KUKA KRL program: MyProgram_237().src

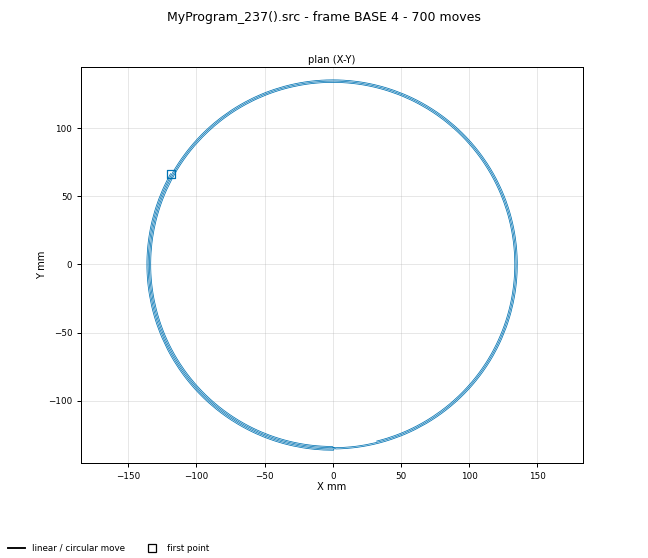
[picture p0: tool path of MyProgram_237().src in frame BASE 4, 700 of 700 moves have a stored position in this frame; points joined in program order, loops and branches not executed]
&ACCESS RVP
&REL 1
&PARAM TEMPLATE = C:\KRC\Roboter\Template\vorgabe
&PARAM EDITMASK = *
DEF MyProgram_237()
; ---- Setting reference (Base) ----
$BASE = BASE_DATA[4]

; --------------------------
; ---- Setting tool (TCP) ----
$TOOL = TOOL_DATA[3]
; --------------------------

$VEL.CP = VEL_APROX_PRINT
Startdeposition()
$VEL.CP = VEL_PRINT
LIN {X -118.9926,Y 66.6239,Z 160,A 148.5784,B 23.5572,C -1.283,E1 23.449,E2 298.3688} C_DIS
LIN {X -121.2876,Y 62.3465,Z 160,A 150.2313,B 23.5584,C -1.2585,E1 23.447,E2 296.7681} C_DIS
LIN {X -123.5569,Y 57.7188,Z 160,A 152.2779,B 23.5591,C -1.2464,E1 23.4445,E2 294.7403} C_DIS
LIN {X -125.0146,Y 54.4885,Z 160,A 153.7,B 23.5594,C -1.2386,E1 23.4429,E2 293.3293} C_DIS
LIN {X -126.4544,Y 51.0566,Z 160,A 155.2792,B 23.5596,C -1.2346,E1 23.4412,E2 291.751} C_DIS
LIN {X -127.5918,Y 48.145,Z 160,A 156.5985,B 23.5598,C -1.2307,E1 23.4399,E2 290.4334} C_DIS
LIN {X -128.7443,Y 44.9722,Z 160,A 158.0153,B 23.5601,C -1.2262,E1 23.4386,E2 289.0194} C_DIS
LIN {X -129.5584,Y 42.5724,Z 160,A 159.5184,B 23.5592,C -1.2435,E1 23.4373,E2 287.4635} C_DIS
LIN {X -130.7224,Y 38.8522,Z 160,A 160.8124,B 23.5603,C -1.2221,E1 23.4362,E2 286.2155} C_DIS
LIN {X -131.707,Y 35.3675,Z 160,A 162.2633,B 23.5607,C -1.2139,E1 23.4352,E2 284.7762} C_DIS
LIN {X -132.5011,Y 32.2662,Z 160,A 163.6223,B 23.5608,C -1.2102,E1 23.4342,E2 283.4179} C_DIS
LIN {X -133.2335,Y 29.0944,Z 160,A 165.0699,B 23.5608,C -1.2096,E1 23.4334,E2 281.9629} C_DIS
LIN {X -134.0169,Y 25.2423,Z 160,A 166.7918,B 23.561,C -1.2075,E1 23.4324,E2 280.2352} C_DIS
LIN {X -134.7535,Y 20.9542,Z 160,A 168.5433,B 23.5614,C -1.198,E1 23.4317,E2 278.4967} C_DIS
LIN {X -135.3189,Y 16.9412,Z 160,A 170.3698,B 23.5614,C -1.1982,E1 23.431,E2 276.658} C_DIS
LIN {X -135.712,Y 13.4163,Z 160,A 171.719,B 23.562,C -1.1867,E1 23.4306,E2 275.329} C_DIS
LIN {X -136.0044,Y 10.0208,Z 160,A 173.2395,B 23.562,C -1.1862,E1 23.4303,E2 273.8} C_DIS
LIN {X -136.2543,Y 5.7048,Z 160,A 175.0307,B 23.5623,C -1.1791,E1 23.43,E2 272.0153} C_DIS
LIN {X -136.3568,Y 2.1131,Z 160,A 176.588,B 23.5624,C -1.1764,E1 23.43,E2 270.4546} C_DIS
LIN {X -136.3514,Y -2.4394,Z 160,A 178.4811,B 23.5628,C -1.1693,E1 23.43,E2 268.5674} C_DIS
LIN {X -136.2184,Y -6.5022,Z 160,A -179.7767,B 23.563,C -1.1653,E1 23.4302,E2 266.8239} C_DIS
LIN {X -135.9819,Y -10.3286,Z 160,A -178.1684,B 23.5632,C -1.16,E1 23.4305,E2 265.2187} C_DIS
LIN {X -135.6069,Y -14.4357,Z 160,A -176.4169,B 23.5634,C -1.1553,E1 23.4309,E2 263.4679} C_DIS
LIN {X -135.1517,Y -18.2164,Z 160,A -174.7244,B 23.5634,C -1.1545,E1 23.4315,E2 261.7665} C_DIS
LIN {X -134.5594,Y -22.1676,Z 160,A -173.1183,B 23.5639,C -1.1457,E1 23.4322,E2 260.1723} C_DIS
LIN {X -132.9907,Y -30.1838,Z 160,A -169.6362,B 23.5643,C -1.1372,E1 23.4342,E2 256.6896} C_DIS
LIN {X -132.0789,Y -33.9538,Z 160,A -167.9215,B 23.5643,C -1.1361,E1 23.4354,E2 254.9669} C_DIS
LIN {X -130.964,Y -38.0269,Z 160,A -166.3432,B 23.565,C -1.1214,E1 23.4365,E2 253.4161} C_DIS
LIN {X -130.0625,Y -41.0063,Z 160,A -164.8722,B 23.5648,C -1.1251,E1 23.4378,E2 251.9266} C_DIS
LIN {X -128.9154,Y -44.4789,Z 160,A -163.3824,B 23.5651,C -1.1182,E1 23.4391,E2 250.445} C_DIS
LIN {X -127.7244,Y -47.7909,Z 160,A -161.9393,B 23.5654,C -1.1121,E1 23.4405,E2 249.0086} C_DIS
LIN {X -126.5403,Y -50.8435,Z 160,A -160.482,B 23.5654,C -1.1119,E1 23.442,E2 247.5431} C_DIS
LIN {X -125.2476,Y -53.9495,Z 160,A -159.1344,B 23.5657,C -1.1047,E1 23.4434,E2 246.2057} C_DIS
LIN {X -121.1191,Y -62.6761,Z 160,A -155.0024,B 23.5661,C -1.0965,E1 23.4485,E2 242.0702} C_DIS
LIN {X -118.6948,Y -67.1543,Z 160,A -152.7589,B 23.5661,C -1.0956,E1 23.4515,E2 239.8165} C_DIS
LIN {X -116.5618,Y -70.7914,Z 160,A -151.0585,B 23.5665,C -1.0874,E1 23.4539,E2 238.1273} C_DIS
LIN {X -112.5394,Y -77.0255,Z 160,A -147.8415,B 23.5666,C -1.084,E1 23.4588,E2 234.9016} C_DIS
LIN {X -109.8378,Y -80.8311,Z 160,A -145.9935,B 23.5671,C -1.0736,E1 23.4618,E2 233.0701} C_DIS
LIN {X -107.641,Y -83.7346,Z 160,A -144.404,B 23.5671,C -1.0728,E1 23.4645,E2 231.4747} C_DIS
LIN {X -104.9293,Y -87.1084,Z 160,A -142.6985,B 23.5675,C -1.0629,E1 23.4675,E2 229.7855} C_DIS
LIN {X -101.6155,Y -90.9522,Z 160,A -140.3512,B 23.5673,C -1.0684,E1 23.4719,E2 227.4131} C_DIS
LIN {X -98.4957,Y -94.3219,Z 160,A -138.5662,B 23.5678,C -1.0571,E1 23.4753,E2 225.6482} C_DIS
LIN {X -94.701,Y -98.1314,Z 160,A -136.1362,B 23.5676,C -1.0605,E1 23.4801,E2 223.1987} C_DIS
LIN {X -91.0992,Y -101.4838,Z 160,A -133.1464,B 23.5658,C -1.1018,E1 23.4866,E2 220.0923} C_DIS
LIN {X -85.5869,Y -106.1739,Z 160,A -131.0457,B 23.5681,C -1.0495,E1 23.4908,E2 218.1147} C_DIS
LIN {X -81.7858,Y -109.1296,Z 160,A -129.0308,B 23.5683,C -1.0454,E1 23.4953,E2 216.1021} C_DIS
LIN {X -78.2738,Y -111.6754,Z 160,A -127.1485,B 23.5683,C -1.0452,E1 23.4996,E2 214.2134} C_DIS
LIN {X -74.6255,Y -114.1456,Z 160,A -125.3166,B 23.5684,C -1.0412,E1 23.5038,E2 212.385} C_DIS
LIN {X -69.3964,Y -117.398,Z 160,A -122.6893,B 23.5685,C -1.0393,E1 23.5101,E2 209.7539} C_DIS
LIN {X -66.0931,Y -119.2884,Z 160,A -121.1313,B 23.5687,C -1.035,E1 23.5139,E2 208.2019} C_DIS
LIN {X -62.2401,Y -121.3417,Z 160,A -119.3539,B 23.5689,C -1.0298,E1 23.5183,E2 206.4324} C_DIS
LIN {X -59.0874,Y -122.9075,Z 160,A -117.8743,B 23.5689,C -1.028,E1 23.522,E2 204.9531} C_DIS
LIN {X -55.9819,Y -124.3528,Z 160,A -116.6382,B 23.5695,C -1.0162,E1 23.5251,E2 203.7433} C_DIS
LIN {X -50.5222,Y -126.6698,Z 160,A -113.9638,B 23.5692,C -1.0226,E1 23.532,E2 201.0463} C_DIS
LIN {X -46.435,Y -128.2237,Z 160,A -112.0439,B 23.5692,C -1.025,E1 23.5371,E2 199.1161} C_DIS
LIN {X -42.7262,Y -129.5072,Z 160,A -110.3745,B 23.5692,C -1.0247,E1 23.5415,E2 197.4442} C_DIS
LIN {X -38.5738,Y -130.8039,Z 160,A -108.6083,B 23.5693,C -1.0202,E1 23.5462,E2 195.686} C_DIS
LIN {X -35.2796,Y -131.7304,Z 160,A -107.2059,B 23.5694,C -1.0175,E1 23.5499,E2 194.2881} C_DIS
LIN {X -31.7741,Y -132.6197,Z 160,A -105.6159,B 23.5694,C -1.0202,E1 23.5543,E2 192.689} C_DIS
LIN {X -28.5037,Y -133.361,Z 160,A -103.3189,B 23.5674,C -1.0649,E1 23.5609,E2 190.277} C_DIS
LIN {X -21.8819,Y -134.6071,Z 160,A -101.3405,B 23.5693,C -1.0202,E1 23.566,E2 188.4086} C_DIS
LIN {X -17.9115,Y -135.1917,Z 160,A -99.972,B 23.57,C -1.0037,E1 23.5697,E2 187.0802} C_DIS
LIN {X -12.7092,Y -135.7799,Z 160,A -96.6912,B 23.5677,C -1.0589,E1 23.5792,E2 183.6593} C_DIS
LIN {X -6.5196,Y -136.2175,Z 160,A -94.9524,B 23.5696,C -1.0141,E1 23.5837,E2 182.0318} C_DIS
LIN {X 0.6255,Y -136.3718,Z 160,A -92.0832,B 23.5698,C -1.0077,E1 23.5917,E2 179.1785} C_DIS
LIN {X 0.6255,Y -136.3718,Z 160,A -92.0832,B 23.5698,C -1.0077,E1 23.5917,E2 179.1785} C_DIS
Enddeposition()
LIN {X 0.9621,Y -135.4362,Z 160,A -91.6873,B 21.9641,C -0.7399,E1 21.9772,E2 179.2938} C_DIS
Startdeposition()
$VEL.CP = VEL_PRINT
LIN {X -3.6024,Y -135.3994,Z 160,A -93.5739,B 21.9641,C -0.7415,E1 21.9719,E2 181.1761} C_DIS
LIN {X -6.6447,Y -135.2842,Z 160,A -95.1252,B 21.9644,C -0.7291,E1 21.9675,E2 182.761} C_DIS
LIN {X -10.3175,Y -135.0544,Z 160,A -96.9624,B 21.9649,C -0.7161,E1 21.9623,E2 184.6339} C_DIS
LIN {X -13.5627,Y -134.7677,Z 160,A -98.238,B 21.9647,C -0.721,E1 21.9587,E2 185.8972} C_DIS
LIN {X -17.8068,Y -134.2716,Z 160,A -99.829,B 21.9644,C -0.7314,E1 21.9544,E2 187.4617} C_DIS
LIN {X -21.1498,Y -133.7863,Z 160,A -101.2751,B 21.9644,C -0.731,E1 21.9504,E2 188.9102} C_DIS
LIN {X -24.2668,Y -133.256,Z 160,A -102.9482,B 21.9649,C -0.716,E1 21.9457,E2 190.6255} C_DIS
LIN {X -27.6501,Y -132.5963,Z 160,A -104.0571,B 21.9643,C -0.7327,E1 21.9428,E2 191.6912} C_DIS
LIN {X -30.692,Y -131.9248,Z 160,A -105.4462,B 21.9644,C -0.7301,E1 21.939,E2 193.0893} C_DIS
LIN {X -34.7695,Y -130.9082,Z 160,A -107.2187,B 21.9644,C -0.7314,E1 21.9342,E2 194.8612} C_DIS
LIN {X -38.1022,Y -129.9772,Z 160,A -108.6616,B 21.9644,C -0.7333,E1 21.9303,E2 196.3015} C_DIS
LIN {X -41.3625,Y -128.9767,Z 160,A -110.1289,B 21.9644,C -0.7333,E1 21.9264,E2 197.7719} C_DIS
LIN {X -45.0409,Y -127.7405,Z 160,A -112.0238,B 21.9646,C -0.7232,E1 21.9213,E2 199.6982} C_DIS
LIN {X -49.2765,Y -126.1653,Z 160,A -113.6914,B 21.9642,C -0.7361,E1 21.917,E2 201.3352} C_DIS
LIN {X -55.4887,Y -123.5591,Z 160,A -116.5223,B 21.9641,C -0.74,E1 21.9098,E2 204.1632} C_DIS
LIN {X -58.5818,Y -122.1229,Z 160,A -117.9831,B 21.9641,C -0.7409,E1 21.9061,E2 205.626} C_DIS
LIN {X -61.723,Y -120.566,Z 160,A -119.474,B 21.9641,C -0.7424,E1 21.9024,E2 207.1174} C_DIS
LIN {X -65.1604,Y -118.7458,Z 160,A -121.2225,B 21.9641,C -0.7399,E1 21.898,E2 208.8782} C_DIS
LIN {X -69.084,Y -116.506,Z 160,A -123.512,B 21.9645,C -0.7258,E1 21.8924,E2 211.2135} C_DIS
LIN {X -72.7665,Y -114.243,Z 160,A -124.6697,B 21.9635,C -0.7585,E1 21.8899,E2 212.2876} C_DIS
LIN {X -75.1993,Y -112.6561,Z 160,A -126.1897,B 21.9639,C -0.7475,E1 21.8862,E2 213.8431} C_DIS
LIN {X -78.8618,Y -110.1234,Z 160,A -128.0645,B 21.9637,C -0.751,E1 21.882,E2 215.7158} C_DIS
LIN {X -82.5025,Y -107.4231,Z 160,A -130.0066,B 21.9637,C -0.7533,E1 21.8776,E2 217.6598} C_DIS
LIN {X -85.9062,Y -104.7211,Z 160,A -131.8112,B 21.9635,C -0.7582,E1 21.8737,E2 219.459} C_DIS
LIN {X -90.4175,Y -100.8514,Z 160,A -134.3556,B 21.9634,C -0.7618,E1 21.8684,E2 222.0053} C_DIS
LIN {X -93.6344,Y -97.8719,Z 160,A -136.2177,B 21.9633,C -0.7653,E1 21.8646,E2 223.8669} C_DIS
LIN {X -97.1401,Y -94.3938,Z 160,A -138.3591,B 21.9633,C -0.7675,E1 21.8603,E2 226.0129} C_DIS
LIN {X -100.2567,Y -91.0765,Z 160,A -140.2831,B 21.9631,C -0.7718,E1 21.8567,E2 227.9351} C_DIS
LIN {X -103.4388,Y -87.4464,Z 160,A -142.1169,B 21.9626,C -0.7856,E1 21.8534,E2 229.7413} C_DIS
LIN {X -105.4457,Y -85.0148,Z 160,A -143.6687,B 21.9628,C -0.7792,E1 21.8506,E2 231.3186} C_DIS
LIN {X -108.2907,Y -81.3606,Z 160,A -145.6019,B 21.9626,C -0.7851,E1 21.8473,E2 233.2467} C_DIS
LIN {X -110.878,Y -77.7979,Z 160,A -147.5162,B 21.9626,C -0.7875,E1 21.8442,E2 235.1653} C_DIS
LIN {X -113.242,Y -74.3143,Z 160,A -149.4657,B 21.9626,C -0.7848,E1 21.8412,E2 237.1335} C_DIS
LIN {X -115.5765,Y -70.6289,Z 160,A -151.1544,B 21.9622,C -0.7964,E1 21.8387,E2 238.8009} C_DIS
LIN {X -117.8279,Y -66.806,Z 160,A -153.1467,B 21.9622,C -0.7964,E1 21.8359,E2 240.8051} C_DIS
LIN {X -120.0606,Y -62.7002,Z 160,A -154.9729,B 21.9618,C -0.8084,E1 21.8336,E2 242.6103} C_DIS
LIN {X -121.9143,Y -59.0186,Z 160,A -157.2735,B 21.9625,C -0.7893,E1 21.8307,E2 244.9767} C_DIS
LIN {X -123.878,Y -54.7756,Z 160,A -158.6627,B 21.9614,C -0.8202,E1 21.8292,E2 246.2915} C_DIS
LIN {X -125.0588,Y -52.0206,Z 160,A -159.9812,B 21.9614,C -0.8217,E1 21.8277,E2 247.6144} C_DIS
LIN {X -126.3506,Y -48.7999,Z 160,A -161.4648,B 21.9612,C -0.8253,E1 21.8262,E2 249.098} C_DIS
LIN {X -127.5141,Y -45.6733,Z 160,A -162.8651,B 21.961,C -0.8299,E1 21.8249,E2 250.4949} C_DIS
LIN {X -128.731,Y -42.1266,Z 160,A -164.5953,B 21.961,C -0.8284,E1 21.8233,E2 252.2406} C_DIS
LIN {X -129.9198,Y -38.2981,Z 160,A -166.2639,B 21.9609,C -0.8347,E1 21.822,E2 253.9034} C_DIS
LIN {X -130.9593,Y -34.5776,Z 160,A -167.8267,B 21.9606,C -0.8428,E1 21.8208,E2 255.455} C_DIS
LIN {X -132.0465,Y -30.1591,Z 160,A -170.7115,B 21.9618,C -0.808,E1 21.819,E2 258.4531} C_DIS
LIN {X -133.3797,Y -23.5757,Z 160,A -172.5089,B 21.9599,C -0.8611,E1 21.8181,E2 260.1197} C_DIS
LIN {X -133.8391,Y -20.8086,Z 160,A -173.8181,B 21.9599,C -0.8596,E1 21.8175,E2 261.442} C_DIS
LIN {X -134.3147,Y -17.4777,Z 160,A -175.2975,B 21.9599,C -0.8617,E1 21.8169,E2 262.9261} C_DIS
LIN {X -134.8037,Y -13.1884,Z 160,A -177.1458,B 21.9597,C -0.8665,E1 21.8164,E2 264.7741} C_DIS
LIN {X -135.1311,Y -9.2669,Z 160,A -178.8967,B 21.9597,C -0.8681,E1 21.816,E2 266.5329} C_DIS
LIN {X -135.3485,Y -5.1699,Z 160,A 179.4466,B 21.9593,C -0.8771,E1 21.8158,E2 268.1771} C_DIS
LIN {X -135.4457,Y -0.789,Z 160,A 177.6628,B 21.959,C -0.886,E1 21.8158,E2 269.9493} C_DIS
LIN {X -135.4241,Y 2.5173,Z 160,A 176.1951,B 21.959,C -0.8875,E1 21.8158,E2 271.4231} C_DIS
LIN {X -135.2841,Y 6.6458,Z 160,A 174.4162,B 21.9587,C -0.8918,E1 21.816,E2 273.2028} C_DIS
LIN {X -135.06,Y 10.2409,Z 160,A 172.8421,B 21.9587,C -0.8945,E1 21.8163,E2 274.7805} C_DIS
LIN {X -134.6705,Y 14.4832,Z 160,A 171.1093,B 21.9583,C -0.9033,E1 21.8168,E2 276.5017} C_DIS
LIN {X -134.2709,Y 17.8124,Z 160,A 169.6786,B 21.9581,C -0.9073,E1 21.8173,E2 277.9315} C_DIS
LIN {X -133.724,Y 21.5484,Z 160,A 167.9141,B 21.9582,C -0.9053,E1 21.818,E2 279.7136} C_DIS
LIN {X -133.0318,Y 25.4642,Z 160,A 166.3272,B 21.9578,C -0.9147,E1 21.8188,E2 281.286} C_DIS
LIN {X -132.1863,Y 29.5473,Z 160,A 164.4073,B 21.9578,C -0.9137,E1 21.8199,E2 283.2218} C_DIS
LIN {X -131.2621,Y 33.4084,Z 160,A 162.8919,B 21.9574,C -0.926,E1 21.8209,E2 284.7143} C_DIS
LIN {X -130.1663,Y 37.4562,Z 160,A 160.6198,B 21.958,C -0.9104,E1 21.8227,E2 287.0436} C_DIS
LIN {X -128.9607,Y 41.4127,Z 160,A 159.3216,B 21.957,C -0.935,E1 21.8238,E2 288.2841} C_DIS
LIN {X -127.974,Y 44.3677,Z 160,A 158.0167,B 21.9568,C -0.9396,E1 21.8249,E2 289.5853} C_DIS
LIN {X -126.7763,Y 47.6825,Z 160,A 156.5194,B 21.9567,C -0.9439,E1 21.8264,E2 291.0807} C_DIS
LIN {X -125.5135,Y 50.9143,Z 160,A 155.041,B 21.9565,C -0.9479,E1 21.8279,E2 292.5579} C_DIS
LIN {X -124.2359,Y 53.9564,Z 160,A 153.597,B 21.9565,C -0.9501,E1 21.8295,E2 294.0053} C_DIS
LIN {X -122.6045,Y 57.5724,Z 160,A 151.6607,B 21.9567,C -0.9441,E1 21.8318,E2 295.9701} C_DIS
LIN {X -120.4337,Y 61.9828,Z 160,A 149.8245,B 21.956,C -0.9606,E1 21.834,E2 297.7732} C_DIS
LIN {X -117.8067,Y 66.8432,Z 160,A 147.3938,B 21.9559,C -0.9633,E1 21.8373,E2 300.2113} C_DIS
LIN {X -115.6401,Y 70.5253,Z 160,A 145.5271,B 21.9558,C -0.9659,E1 21.84,E2 302.0822} C_DIS
LIN {X -113.1582,Y 74.4416,Z 160,A 143.2602,B 21.9561,C -0.9584,E1 21.8435,E2 304.3827} C_DIS
LIN {X -110.9089,Y 77.754,Z 160,A 142.1606,B 21.9548,C -0.9884,E1 21.8452,E2 305.4077} C_DIS
LIN {X -107.9092,Y 81.8661,Z 160,A 139.6213,B 21.9553,C -0.9776,E1 21.8494,E2 307.9903} C_DIS
LIN {X -105.2413,Y 85.2682,Z 160,A 137.3826,B 21.9558,C -0.9648,E1 21.8534,E2 310.2753} C_DIS
LIN {X -102.1389,Y 88.9605,Z 160,A 135.9969,B 21.9544,C -0.9981,E1 21.8558,E2 311.5789} C_DIS
LIN {X -99.6611,Y 91.7278,Z 160,A 134.2543,B 21.9545,C -0.9946,E1 21.8591,E2 313.3398} C_DIS
LIN {X -96.5021,Y 95.0461,Z 160,A 132.3015,B 21.9544,C -0.9987,E1 21.8629,E2 315.2915} C_DIS
LIN {X -93.3021,Y 98.1896,Z 160,A 130.3884,B 21.9542,C -1.0025,E1 21.8667,E2 317.2035} C_DIS
LIN {X -90.0635,Y 101.1684,Z 160,A 128.5201,B 21.954,C -1.0064,E1 21.8706,E2 319.0699} C_DIS
LIN {X -86.7543,Y 104.0201,Z 160,A 125.8575,B 21.9554,C -0.9753,E1 21.8765,E2 321.8278} C_DIS
LIN {X -81.7211,Y 108.0185,Z 160,A 124.1711,B 21.9532,C -1.0257,E1 21.88,E2 323.386} C_DIS
LIN {X -74.5587,Y 113.0811,Z 160,A 120.1563,B 21.9534,C -1.0196,E1 21.8892,E2 327.4329} C_DIS
LIN {X -71.1893,Y 115.2326,Z 160,A 118.4924,B 21.9533,C -1.0239,E1 21.8931,E2 329.0914} C_DIS
LIN {X -67.4456,Y 117.463,Z 160,A 116.6616,B 21.9531,C -1.0277,E1 21.8975,E2 330.9183} C_DIS
LIN {X -63.8987,Y 119.4292,Z 160,A 114.9581,B 21.9529,C -1.0311,E1 21.9017,E2 332.6183} C_DIS
LIN {X -59.1266,Y 121.8627,Z 160,A 112.7618,B 21.9526,C -1.0378,E1 21.9072,E2 334.8034} C_DIS
LIN {X -56.6,Y 123.0541,Z 160,A 111.5172,B 21.9526,C -1.0368,E1 21.9103,E2 336.0541} C_DIS
LIN {X -52.5123,Y 124.8534,Z 160,A 109.4998,B 21.9528,C -1.0339,E1 21.9155,E2 338.085} C_DIS
LIN {X -49.0701,Y 126.2456,Z 160,A 108.0641,B 21.9525,C -1.0419,E1 21.9192,E2 339.5027} C_DIS
LIN {X -45.7417,Y 127.4895,Z 160,A 106.6127,B 21.9523,C -1.0461,E1 21.923,E2 340.9462} C_DIS
LIN {X -42.5303,Y 128.5966,Z 160,A 105.1147,B 21.9523,C -1.0451,E1 21.927,E2 342.4502} C_DIS
LIN {X -35.6562,Y 130.6717,Z 160,A 102.1237,B 21.9521,C -1.0504,E1 21.935,E2 345.4328} C_DIS
LIN {X -31.5859,Y 131.7126,Z 160,A 100.2958,B 21.9521,C -1.0498,E1 21.9399,E2 347.2652} C_DIS
LIN {X -27.3973,Y 132.6477,Z 160,A 98.4634,B 21.9521,C -1.0506,E1 21.9449,E2 349.0983} C_DIS
LIN {X -23.7948,Y 133.3405,Z 160,A 96.9896,B 21.9518,C -1.0552,E1 21.949,E2 350.5612} C_DIS
LIN {X -20.6085,Y 133.8701,Z 160,A 95.5687,B 21.9519,C -1.0537,E1 21.9529,E2 351.9878} C_DIS
LIN {X -17.0008,Y 134.3772,Z 160,A 93.9024,B 21.9521,C -1.0489,E1 21.9575,E2 353.6683} C_DIS
LIN {X -12.6352,Y 134.8568,Z 160,A 92.1536,B 21.9519,C -1.0548,E1 21.9624,E2 355.4026} C_DIS
LIN {X -8.3244,Y 135.1911,Z 160,A 90.3503,B 21.9518,C -1.0567,E1 21.9674,E2 357.2016} C_DIS
LIN {X -4.4468,Y 135.3759,Z 160,A 88.5636,B 21.9521,C -1.0506,E1 21.9724,E2 359.0051} C_DIS
LIN {X 0.0544,Y 135.449,Z 160,A 86.661,B 21.9521,C -1.051,E1 21.9777,E2 360.9065} C_DIS
LIN {X 3.8844,Y 135.3915,Z 160,A 85.1395,B 21.9518,C -1.0557,E1 21.9819,E2 362.4151} C_DIS
LIN {X 8.0031,Y 135.2109,Z 160,A 83.2602,B 21.9521,C -1.0495,E1 21.9872,E2 364.3103} C_DIS
LIN {X 13.1417,Y 134.8082,Z 160,A 81.2144,B 21.9518,C -1.0554,E1 21.9929,E2 366.3389} C_DIS
LIN {X 17.6346,Y 134.2942,Z 160,A 79.2629,B 21.9519,C -1.0532,E1 21.9983,E2 368.2945} C_DIS
LIN {X 21.6033,Y 133.7149,Z 160,A 77.4061,B 21.9523,C -1.0453,E1 22.0035,E2 370.1705} C_DIS
LIN {X 26.0559,Y 132.9187,Z 160,A 75.5996,B 21.9521,C -1.0494,E1 22.0084,E2 371.9637} C_DIS
LIN {X 30.0594,Y 132.0693,Z 160,A 73.9772,B 21.9519,C -1.0535,E1 22.0128,E2 373.5724} C_DIS
LIN {X 33.4396,Y 131.2542,Z 160,A 72.5493,B 21.9519,C -1.0546,E1 22.0166,E2 374.995} C_DIS
LIN {X 36.6391,Y 130.3973,Z 160,A 71.1278,B 21.9519,C -1.0527,E1 22.0204,E2 376.4189} C_DIS
LIN {X 40.1258,Y 129.3678,Z 160,A 69.5912,B 21.952,C -1.0516,E1 22.0246,E2 377.9553} C_DIS
LIN {X 45.1696,Y 127.6957,Z 160,A 67.366,B 21.952,C -1.0507,E1 22.0304,E2 380.178} C_DIS
LIN {X 52.3518,Y 124.9205,Z 160,A 64.1027,B 21.9522,C -1.0471,E1 22.0389,E2 383.4425} C_DIS
LIN {X 55.4472,Y 123.5776,Z 160,A 62.6685,B 21.9523,C -1.0451,E1 22.0426,E2 384.8779} C_DIS
LIN {X 58.6262,Y 122.1017,Z 160,A 61.1812,B 21.9523,C -1.0431,E1 22.0463,E2 386.3661} C_DIS
LIN {X 61.8215,Y 120.5158,Z 160,A 59.6981,B 21.9524,C -1.0424,E1 22.05,E2 387.8466} C_DIS
LIN {X 65.2203,Y 118.7131,Z 160,A 57.957,B 21.9528,C -1.0347,E1 22.0544,E2 389.6023} C_DIS
LIN {X 69.1222,Y 116.484,Z 160,A 56.0779,B 21.9528,C -1.0329,E1 22.0589,E2 391.4794} C_DIS
LIN {X 72.8604,Y 114.1829,Z 160,A 54.2455,B 21.9529,C -1.0312,E1 22.0632,E2 393.3098} C_DIS
LIN {X 76.4861,Y 111.7866,Z 160,A 52.3879,B 21.9531,C -1.0273,E1 22.0675,E2 395.1706} C_DIS
LIN {X 80.3614,Y 109.034,Z 160,A 50.5718,B 21.9528,C -1.0331,E1 22.0716,E2 396.9639} C_DIS
LIN {X 83.2733,Y 106.8271,Z 160,A 48.0827,B 21.9549,C -0.9853,E1 22.0773,E2 399.5697} C_DIS
LIN {X 88.1924,Y 102.8032,Z 160,A 46.3323,B 21.9532,C -1.0248,E1 22.0808,E2 401.2069} C_DIS
LIN {X 90.926,Y 100.3933,Z 160,A 44.6612,B 21.9536,C -1.0155,E1 22.0843,E2 402.8953} C_DIS
LIN {X 94.8811,Y 96.6639,Z 160,A 42.7284,B 21.9531,C -1.0284,E1 22.0882,E2 404.7845} C_DIS
LIN {X 97.6299,Y 93.8877,Z 160,A 40.6857,B 21.9541,C -1.0059,E1 22.0923,E2 406.877} C_DIS
LIN {X 101.7299,Y 89.4287,Z 160,A 38.2535,B 21.9541,C -1.0064,E1 22.0968,E2 409.2954} C_DIS
LIN {X 104.372,Y 86.3297,Z 160,A 36.4603,B 21.9544,C -0.9989,E1 22.1,E2 411.099} C_DIS
LIN {X 107.206,Y 82.7844,Z 160,A 34.5509,B 21.9545,C -0.9948,E1 22.1033,E2 413.009} C_DIS
LIN {X 109.9242,Y 79.1402,Z 160,A 31.9269,B 21.9562,C -0.956,E1 22.1078,E2 415.7214} C_DIS
LIN {X 113.3162,Y 74.2015,Z 160,A 30.1356,B 21.9549,C -0.9855,E1 22.1104,E2 417.424} C_DIS
LIN {X 115.6843,Y 70.4532,Z 160,A 28.2272,B 21.9552,C -0.979,E1 22.1132,E2 419.3386} C_DIS
LIN {X 117.9534,Y 66.5838,Z 160,A 26.3474,B 21.9554,C -0.9747,E1 22.1158,E2 421.2186} C_DIS
LIN {X 120.0672,Y 62.6878,Z 160,A 24.593,B 21.9554,C -0.9755,E1 22.1181,E2 422.9602} C_DIS
LIN {X 121.5296,Y 59.8027,Z 160,A 23.2355,B 21.9554,C -0.9722,E1 22.1198,E2 424.3181} C_DIS
LIN {X 123.0606,Y 56.5858,Z 160,A 21.7446,B 21.9556,C -0.9687,E1 22.1216,E2 425.8089} C_DIS
LIN {X 124.3792,Y 53.625,Z 160,A 20.3817,B 21.9558,C -0.9652,E1 22.1231,E2 427.1726} C_DIS
LIN {X 125.7532,Y 50.3195,Z 160,A 18.7788,B 21.9562,C -0.9564,E1 22.1248,E2 428.7887} C_DIS
LIN {X 127.1636,Y 46.6454,Z 160,A 17.1142,B 21.9564,C -0.9515,E1 22.1265,E2 430.4557} C_DIS
LIN {X 128.9475,Y 41.4541,Z 160,A 14.5207,B 21.9572,C -0.9312,E1 22.1288,E2 433.0862} C_DIS
LIN {X 130.073,Y 37.7751,Z 160,A 13.3187,B 21.9565,C -0.9472,E1 22.1297,E2 434.2376} C_DIS
LIN {X 130.975,Y 34.5191,Z 160,A 11.7596,B 21.957,C -0.9364,E1 22.1308,E2 435.8151} C_DIS
LIN {X 132.0121,Y 30.3097,Z 160,A 10.0128,B 21.957,C -0.9351,E1 22.1319,E2 437.5537} C_DIS
LIN {X 132.7768,Y 26.763,Z 160,A 8.5324,B 21.9571,C -0.933,E1 22.1328,E2 439.0297} C_DIS
LIN {X 133.5293,Y 22.7156,Z 160,A 6.7512,B 21.9574,C -0.9256,E1 22.1337,E2 440.8186} C_DIS
LIN {X 134.0985,Y 19.0657,Z 160,A 5.2345,B 21.9575,C -0.9229,E1 22.1343,E2 442.3321} C_DIS
LIN {X 134.6344,Y 14.8184,Z 160,A 3.4079,B 21.9578,C -0.9164,E1 22.1349,E2 444.1636} C_DIS
LIN {X 134.9855,Y 11.1757,Z 160,A 1.9516,B 21.9578,C -0.916,E1 22.1353,E2 445.6108} C_DIS
LIN {X 135.3137,Y 6.0543,Z 160,A -0.1724,B 21.958,C -0.9114,E1 22.1356,E2 447.7326} C_DIS
LIN {X 135.438,Y 1.6818,Z 160,A -2.0292,B 21.9582,C -0.9051,E1 22.1357,E2 449.5932} C_DIS
LIN {X 135.4206,Y -2.7263,Z 160,A -3.9036,B 21.9585,C -0.8986,E1 22.1357,E2 451.4721} C_DIS
LIN {X 135.3312,Y -5.6134,Z 160,A -5.2414,B 21.9588,C -0.8889,E1 22.1355,E2 452.8264} C_DIS
LIN {X 135.0829,Y -9.9261,Z 160,A -6.9508,B 21.9588,C -0.8889,E1 22.1352,E2 454.5241} C_DIS
LIN {X 134.7869,Y -13.3631,Z 160,A -8.3674,B 21.9589,C -0.8863,E1 22.1349,E2 455.9379} C_DIS
LIN {X 134.3342,Y -17.3291,Z 160,A -10.1624,B 21.9594,C -0.8756,E1 22.1343,E2 457.7492} C_DIS
LIN {X 133.8352,Y -20.8335,Z 160,A -11.5719,B 21.9594,C -0.8752,E1 22.1337,E2 459.1502} C_DIS
LIN {X 133.2551,Y -24.2722,Z 160,A -13.1368,B 21.9597,C -0.866,E1 22.1329,E2 460.729} C_DIS
LIN {X 132.4172,Y -28.488,Z 160,A -14.8303,B 21.9597,C -0.8664,E1 22.132,E2 462.41} C_DIS
LIN {X 131.6464,Y -31.8606,Z 160,A -16.2421,B 21.9597,C -0.8643,E1 22.1311,E2 463.8178} C_DIS
LIN {X 130.8612,Y -34.9456,Z 160,A -17.6089,B 21.96,C -0.859,E1 22.1301,E2 465.1896} C_DIS
LIN {X 129.8924,Y -38.3919,Z 160,A -19.1189,B 21.9601,C -0.8545,E1 22.1289,E2 466.7017} C_DIS
LIN {X 128.3314,Y -43.3267,Z 160,A -21.2591,B 21.9603,C -0.8501,E1 22.1271,E2 468.8395} C_DIS
LIN {X 127.2422,Y -46.4275,Z 160,A -23.545,B 21.962,C -0.8015,E1 22.1248,E2 471.2397} C_DIS
LIN {X 124.9157,Y -52.3633,Z 160,A -24.9813,B 21.9601,C -0.8557,E1 22.1235,E2 472.5229} C_DIS
LIN {X 123.9701,Y -54.5686,Z 160,A -26.3438,B 21.9609,C -0.8352,E1 22.1219,E2 473.9312} C_DIS
LIN {X 122.1961,Y -58.4287,Z 160,A -28.1787,B 21.9611,C -0.828,E1 22.1197,E2 475.7739} C_DIS
LIN {X 120.5456,Y -61.763,Z 160,A -29.761,B 21.9613,C -0.8229,E1 22.1177,E2 477.36} C_DIS
LIN {X 117.5967,Y -67.2113,Z 160,A -32.3799,B 21.9616,C -0.8153,E1 22.1142,E2 479.9833} C_DIS
LIN {X 115.3356,Y -71.0216,Z 160,A -34.3704,B 21.962,C -0.8042,E1 22.1113,E2 481.9916} C_DIS
LIN {X 112.9678,Y -74.7306,Z 160,A -36.526,B 21.9626,C -0.7845,E1 22.1079,E2 484.1871} C_DIS
LIN {X 110.4301,Y -78.4328,Z 160,A -37.9047,B 21.9619,C -0.8049,E1 22.1058,E2 485.5039} C_DIS
LIN {X 108.1806,Y -81.5065,Z 160,A -39.5989,B 21.9622,C -0.7964,E1 22.103,E2 487.2111} C_DIS
LIN {X 105.3667,Y -85.1129,Z 160,A -41.4989,B 21.9623,C -0.793,E1 22.0997,E2 489.1098} C_DIS
LIN {X 102.5953,Y -88.4337,Z 160,A -43.3293,B 21.9625,C -0.7883,E1 22.0964,E2 490.9432} C_DIS
LIN {X 99.6772,Y -91.7103,Z 160,A -45.1646,B 21.9626,C -0.7846,E1 22.0929,E2 492.7789} C_DIS
LIN {X 96.7166,Y -94.8273,Z 160,A -46.9891,B 21.9628,C -0.7798,E1 22.0894,E2 494.607} C_DIS
LIN {X 93.4467,Y -98.0514,Z 160,A -48.9063,B 21.9629,C -0.7764,E1 22.0855,E2 496.524} C_DIS
LIN {X 90.2754,Y -100.9787,Z 160,A -50.7162,B 21.963,C -0.773,E1 22.0818,E2 498.3346} C_DIS
LIN {X 86.8564,Y -103.9344,Z 160,A -52.6312,B 21.9632,C -0.7685,E1 22.0777,E2 500.2528} C_DIS
LIN {X 83.3764,Y -106.7466,Z 160,A -54.4922,B 21.9632,C -0.766,E1 22.0736,E2 502.1126} C_DIS
LIN {X 79.8529,Y -109.4076,Z 160,A -56.3728,B 21.9634,C -0.7615,E1 22.0694,E2 503.9974} C_DIS
LIN {X 76.271,Y -111.9341,Z 160,A -58.2494,B 21.9636,C -0.7567,E1 22.0651,E2 505.8794} C_DIS
LIN {X 72.4811,Y -114.4241,Z 160,A -60.5649,B 21.9643,C -0.7338,E1 22.0595,E2 508.2472} C_DIS
LIN {X 68.6331,Y -116.7725,Z 160,A -61.6295,B 21.9631,C -0.7711,E1 22.0573,E2 509.2085} C_DIS
LIN {X 60.663,Y -121.1052,Z 160,A -65.7493,B 21.9638,C -0.7507,E1 22.0471,E2 513.3691} C_DIS
LIN {X 57.3727,Y -122.6968,Z 160,A -67.3782,B 21.964,C -0.7443,E1 22.0429,E2 515.0102} C_DIS
LIN {X 53.9219,Y -124.2508,Z 160,A -68.9812,B 21.964,C -0.7418,E1 22.0388,E2 516.6152} C_DIS
LIN {X 50.1985,Y -125.802,Z 160,A -70.6361,B 21.964,C -0.7418,E1 22.0345,E2 518.2656} C_DIS
LIN {X 45.8428,Y -127.453,Z 160,A -72.5073,B 21.964,C -0.7441,E1 22.0296,E2 520.1264} C_DIS
LIN {X 43.3134,Y -128.3358,Z 160,A -73.9588,B 21.9645,C -0.7274,E1 22.0257,E2 521.619} C_DIS
LIN {X 38.5101,Y -129.8577,Z 160,A -76.3531,B 21.965,C -0.7125,E1 22.0192,E2 524.0481} C_DIS
LIN {X 34.0363,Y -131.1027,Z 160,A -77.7321,B 21.9642,C -0.7383,E1 22.0157,E2 525.3558} C_DIS
LIN {X 29.9249,Y -132.1,Z 160,A -79.5643,B 21.9642,C -0.7346,E1 22.0107,E2 527.1949} C_DIS
LIN {X 25.922,Y -132.9443,Z 160,A -81.4004,B 21.9645,C -0.7281,E1 22.0056,E2 529.0458} C_DIS
LIN {X 22.1932,Y -133.6165,Z 160,A -82.9092,B 21.9644,C -0.7314,E1 22.0015,E2 530.5439} C_DIS
LIN {X 17.9687,Y -134.2504,Z 160,A -84.8233,B 21.9646,C -0.7251,E1 21.9962,E2 532.4728} C_DIS
LIN {X 14.5153,Y -134.6671,Z 160,A -86.211,B 21.9645,C -0.7282,E1 21.9923,E2 533.8511} C_DIS
LIN {X 9.65,Y -135.1031,Z 160,A -88.2268,B 21.9645,C -0.7296,E1 21.9867,E2 535.8619} C_DIS
LIN {X 5.6974,Y -135.3279,Z 160,A -89.9402,B 21.9645,C -0.7272,E1 21.9819,E2 537.5811} C_DIS
LIN {X 2.1532,Y -135.4301,Z 160,A -91.6285,B 21.9648,C -0.7179,E1 21.9772,E2 539.2938} C_DIS
LIN {X 2.1532,Y -135.4301,Z 160,A -91.6285,B 21.9648,C -0.7179,E1 21.9772,E2 539.2938} C_DIS
Enddeposition()
LIN {X 0.9519,Y -134.5171,Z 160,A -91.0299,B 20.8115,C -0.592,E1 20.8217,E2 538.924} C_DIS
Startdeposition()
$VEL.CP = VEL_PRINT
LIN {X 3.706,Y -134.4702,Z 160,A -89.7647,B 20.8114,C -0.5964,E1 20.8253,E2 537.6467} C_DIS
LIN {X 6.8857,Y -134.345,Z 160,A -88.3557,B 20.8113,C -0.5993,E1 20.8293,E2 536.2301} C_DIS
LIN {X 10.7338,Y -134.0936,Z 160,A -86.8436,B 20.8114,C -0.5941,E1 20.8334,E2 534.7335} C_DIS
LIN {X 13.6228,Y -133.8318,Z 160,A -85.4325,B 20.8112,C -0.6026,E1 20.8374,E2 533.2995} C_DIS
LIN {X 16.7064,Y -133.482,Z 160,A -84.218,B 20.8113,C -0.5985,E1 20.8407,E2 532.0976} C_DIS
LIN {X 20.297,Y -132.9814,Z 160,A -82.6632,B 20.8113,C -0.6001,E1 20.845,E2 530.5402} C_DIS
LIN {X 24.4783,Y -132.2776,Z 160,A -80.7948,B 20.8112,C -0.6042,E1 20.8502,E2 528.6627} C_DIS
LIN {X 28.1586,Y -131.5411,Z 160,A -79.3406,B 20.8112,C -0.599,E1 20.8541,E2 527.2252} C_DIS
LIN {X 31.2308,Y -130.8458,Z 160,A -77.9039,B 20.8112,C -0.6046,E1 20.8581,E2 525.7755} C_DIS
LIN {X 33.9409,Y -130.1709,Z 160,A -76.7662,B 20.8112,C -0.6033,E1 20.8612,E2 524.6433} C_DIS
LIN {X 37.0152,Y -129.3306,Z 160,A -75.3853,B 20.8112,C -0.6058,E1 20.8649,E2 523.2583} C_DIS
LIN {X 40.1515,Y -128.3916,Z 160,A -73.9928,B 20.8111,C -0.6073,E1 20.8686,E2 521.8647} C_DIS
LIN {X 43.2827,Y -127.3701,Z 160,A -72.5413,B 20.811,C -0.6112,E1 20.8725,E2 520.4056} C_DIS
LIN {X 46.4057,Y -126.2658,Z 160,A -71.1842,B 20.811,C -0.6105,E1 20.876,E2 519.0538} C_DIS
LIN {X 49.5173,Y -125.0783,Z 160,A -69.7688,B 20.811,C -0.6123,E1 20.8797,E2 517.6374} C_DIS
LIN {X 52.6144,Y -123.8074,Z 160,A -68.2023,B 20.8107,C -0.6208,E1 20.8838,E2 516.0516} C_DIS
LIN {X 55.9856,Y -122.3181,Z 160,A -66.9023,B 20.811,C -0.6107,E1 20.887,E2 514.7837} C_DIS
LIN {X 58.752,Y -121.0155,Z 160,A -65.4124,B 20.8107,C -0.6214,E1 20.8908,E2 513.2688} C_DIS
LIN {X 61.7859,Y -119.495,Z 160,A -63.9418,B 20.8106,C -0.6249,E1 20.8945,E2 511.7933} C_DIS
LIN {X 65.539,Y -117.4784,Z 160,A -62.1393,B 20.8105,C -0.6274,E1 20.8989,E2 509.9902} C_DIS
LIN {X 69.2426,Y -115.3343,Z 160,A -60.3165,B 20.8105,C -0.6306,E1 20.9033,E2 508.1651} C_DIS
LIN {X 72.8903,Y -113.0644,Z 160,A -58.5,B 20.8103,C -0.6334,E1 20.9076,E2 506.3479} C_DIS
LIN {X 76.4756,Y -110.6708,Z 160,A -56.6382,B 20.8102,C -0.6382,E1 20.9119,E2 504.4804} C_DIS
LIN {X 79.9926,Y -108.156,Z 160,A -54.8382,B 20.8102,C -0.64,E1 20.9159,E2 502.6832} C_DIS
LIN {X 83.435,Y -105.5232,Z 160,A -53.0011,B 20.81,C -0.6435,E1 20.92,E2 500.8447} C_DIS
LIN {X 86.7971,Y -102.7755,Z 160,A -51.1312,B 20.8099,C -0.6485,E1 20.924,E2 498.9696} C_DIS
LIN {X 90.0758,Y -99.9144,Z 160,A -49.3185,B 20.8099,C -0.6508,E1 20.9278,E2 497.1594} C_DIS
LIN {X 93.2577,Y -96.9512,Z 160,A -47.4763,B 20.8097,C -0.6546,E1 20.9315,E2 495.3157} C_DIS
LIN {X 96.3457,Y -93.8832,Z 160,A -45.6267,B 20.8096,C -0.6589,E1 20.9352,E2 493.4639} C_DIS
LIN {X 99.3321,Y -90.7176,Z 160,A -43.7912,B 20.8095,C -0.6626,E1 20.9387,E2 491.6278} C_DIS
LIN {X 102.2125,Y -87.4594,Z 160,A -41.9444,B 20.8093,C -0.667,E1 20.942,E2 489.7789} C_DIS
LIN {X 104.9827,Y -84.1141,Z 160,A -40.1072,B 20.8092,C -0.6712,E1 20.9453,E2 487.9404} C_DIS
LIN {X 107.6388,Y -80.6872,Z 160,A -38.245,B 20.809,C -0.6768,E1 20.9484,E2 486.0733} C_DIS
LIN {X 110.1774,Y -77.1847,Z 160,A -36.4444,B 20.809,C -0.6798,E1 20.9514,E2 484.2751} C_DIS
LIN {X 112.5955,Y -73.6125,Z 160,A -34.6276,B 20.8088,C -0.6839,E1 20.9542,E2 482.4578} C_DIS
LIN {X 114.8903,Y -69.9768,Z 160,A -32.796,B 20.8086,C -0.6891,E1 20.9569,E2 480.6233} C_DIS
LIN {X 117.0598,Y -66.2839,Z 160,A -30.9946,B 20.8085,C -0.6932,E1 20.9594,E2 478.8218} C_DIS
LIN {X 118.7038,Y -63.2927,Z 160,A -29.5315,B 20.8084,C -0.6978,E1 20.9613,E2 477.3551} C_DIS
LIN {X 120.2656,Y -60.2722,Z 160,A -28.215,B 20.8084,C -0.6958,E1 20.963,E2 476.0529} C_DIS
LIN {X 121.7447,Y -57.2257,Z 160,A -26.7847,B 20.8083,C -0.6995,E1 20.9647,E2 474.6216} C_DIS
LIN {X 123.1406,Y -54.1565,Z 160,A -25.3606,B 20.8082,C -0.7032,E1 20.9663,E2 473.1966} C_DIS
LIN {X 124.4533,Y -51.0679,Z 160,A -23.9434,B 20.8081,C -0.7069,E1 20.9678,E2 471.7787} C_DIS
LIN {X 125.6825,Y -47.9632,Z 160,A -22.5336,B 20.8079,C -0.7107,E1 20.9692,E2 470.368} C_DIS
LIN {X 126.984,Y -44.3965,Z 160,A -20.9136,B 20.8078,C -0.7158,E1 20.9708,E2 468.7448} C_DIS
LIN {X 127.8912,Y -41.718,Z 160,A -19.7369,B 20.8077,C -0.7181,E1 20.9718,E2 467.5697} C_DIS
LIN {X 128.8714,Y -38.5838,Z 160,A -18.3507,B 20.8076,C -0.7219,E1 20.9729,E2 466.1828} C_DIS
LIN {X 129.8661,Y -35.0839,Z 160,A -16.8313,B 20.8075,C -0.7253,E1 20.9741,E2 464.6645} C_DIS
LIN {X 130.7267,Y -31.7247,Z 160,A -15.3636,B 20.8073,C -0.7295,E1 20.9751,E2 463.1954} C_DIS
LIN {X 131.6605,Y -27.6055,Z 160,A -13.5698,B 20.8071,C -0.7348,E1 20.9761,E2 461.3994} C_DIS
LIN {X 132.2776,Y -24.4783,Z 160,A -12.2248,B 20.8071,C -0.7385,E1 20.9768,E2 460.0537} C_DIS
LIN {X 132.8167,Y -21.3603,Z 160,A -10.8517,B 20.8068,C -0.744,E1 20.9775,E2 458.6752} C_DIS
LIN {X 133.2791,Y -18.2542,Z 160,A -9.5651,B 20.8068,C -0.7458,E1 20.978,E2 457.3927} C_DIS
LIN {X 133.6662,Y -15.1625,Z 160,A -8.2508,B 20.8066,C -0.7494,E1 20.9784,E2 456.0779} C_DIS
LIN {X 134.0277,Y -11.5137,Z 160,A -6.6591,B 20.8064,C -0.7559,E1 20.9788,E2 454.4797} C_DIS
LIN {X 134.2736,Y -8.1601,Z 160,A -5.2452,B 20.8063,C -0.7596,E1 20.9791,E2 453.0658} C_DIS
LIN {X 134.4485,Y -4.4884,Z 160,A -3.7359,B 20.8063,C -0.7618,E1 20.9793,E2 451.5611} C_DIS
LIN {X 134.5151,Y -1.4897,Z 160,A -2.3704,B 20.8059,C -0.7701,E1 20.9793,E2 450.1825} C_DIS
LIN {X 134.5017,Y 2.298,Z 160,A -0.8465,B 20.8059,C -0.771,E1 20.9793,E2 448.6672} C_DIS
LIN {X 134.3896,Y 5.9971,Z 160,A 0.6985,B 20.8058,C -0.7745,E1 20.9791,E2 447.1237} C_DIS
LIN {X 134.2199,Y 9.0317,Z 160,A 1.9854,B 20.8056,C -0.7782,E1 20.9789,E2 445.8357} C_DIS
LIN {X 133.9792,Y 12.0875,Z 160,A 3.4301,B 20.8052,C -0.7889,E1 20.9785,E2 444.3716} C_DIS
LIN {X 133.5779,Y 15.9024,Z 160,A 4.9198,B 20.8053,C -0.7873,E1 20.9781,E2 442.8973} C_DIS
LIN {X 133.154,Y 19.1299,Z 160,A 6.2619,B 20.8053,C -0.7895,E1 20.9776,E2 441.5587} C_DIS
LIN {X 132.6814,Y 22.1715,Z 160,A 7.6056,B 20.805,C -0.7951,E1 20.977,E2 440.2089} C_DIS
LIN {X 132.1161,Y 25.3227,Z 160,A 8.9263,B 20.805,C -0.7973,E1 20.9763,E2 438.8915} C_DIS
LIN {X 131.4844,Y 28.4212,Z 160,A 10.2831,B 20.8048,C -0.8019,E1 20.9755,E2 437.5315} C_DIS
LIN {X 130.7674,Y 31.5561,Z 160,A 11.6316,B 20.8046,C -0.8051,E1 20.9747,E2 436.1837} C_DIS
LIN {X 129.9874,Y 34.6289,Z 160,A 12.9652,B 20.8046,C -0.8084,E1 20.9737,E2 434.8502} C_DIS
LIN {X 128.8714,Y 38.5838,Z 160,A 14.7257,B 20.8043,C -0.8141,E1 20.9724,E2 433.0862} C_DIS
LIN {X 127.8912,Y 41.718,Z 160,A 16.1158,B 20.8042,C -0.8179,E1 20.9712,E2 431.6951} C_DIS
LIN {X 126.8283,Y 44.8454,Z 160,A 17.6565,B 20.8038,C -0.8283,E1 20.9697,E2 430.1359} C_DIS
LIN {X 125.496,Y 48.4427,Z 160,A 18.9443,B 20.8042,C -0.8168,E1 20.9685,E2 428.889} C_DIS
LIN {X 124.4533,Y 51.0679,Z 160,A 20.4418,B 20.8036,C -0.8341,E1 20.9669,E2 427.3533} C_DIS
LIN {X 123.0488,Y 54.3619,Z 160,A 21.9333,B 20.8035,C -0.8369,E1 20.9652,E2 425.864} C_DIS
LIN {X 121.7447,Y 57.2257,Z 160,A 23.1823,B 20.8035,C -0.8364,E1 20.9638,E2 424.6248} C_DIS
LIN {X 120.2656,Y 60.2722,Z 160,A 24.6161,B 20.8033,C -0.84,E1 20.962,E2 423.1904} C_DIS
LIN {X 118.39,Y 63.8767,Z 160,A 26.3598,B 20.8031,C -0.8453,E1 20.9597,E2 421.443} C_DIS
LIN {X 116.4305,Y 67.3818,Z 160,A 28.1048,B 20.8029,C -0.8515,E1 20.9573,E2 419.6916} C_DIS
LIN {X 114.1478,Y 71.1805,Z 160,A 29.9674,B 20.8027,C -0.8553,E1 20.9546,E2 417.8301} C_DIS
LIN {X 111.8922,Y 74.6759,Z 160,A 31.7434,B 20.8025,C -0.86,E1 20.9519,E2 416.0516} C_DIS
LIN {X 109.4382,Y 78.2281,Z 160,A 33.572,B 20.8024,C -0.8642,E1 20.9489,E2 414.2224} C_DIS
LIN {X 106.7522,Y 81.8557,Z 160,A 35.4501,B 20.8023,C -0.8668,E1 20.9458,E2 412.348} C_DIS
LIN {X 104.1743,Y 85.1121,Z 160,A 37.2431,B 20.8021,C -0.8721,E1 20.9426,E2 410.5504} C_DIS
LIN {X 101.2608,Y 88.5586,Z 160,A 39.124,B 20.802,C -0.8746,E1 20.9392,E2 408.673} C_DIS
LIN {X 98.4589,Y 91.6635,Z 160,A 40.9265,B 20.8018,C -0.8796,E1 20.9358,E2 406.8663} C_DIS
LIN {X 95.442,Y 94.8008,Z 160,A 42.7706,B 20.8016,C -0.8831,E1 20.9322,E2 405.0219} C_DIS
LIN {X 92.2987,Y 97.8637,Z 160,A 44.623,B 20.8015,C -0.8862,E1 20.9285,E2 403.1702} C_DIS
LIN {X 89.1128,Y 100.7733,Z 160,A 46.4583,B 20.8014,C -0.8898,E1 20.9247,E2 401.3339} C_DIS
LIN {X 85.783,Y 103.6226,Z 160,A 48.3083,B 20.8012,C -0.8926,E1 20.9207,E2 399.4847} C_DIS
LIN {X 82.3959,Y 106.3357,Z 160,A 50.1565,B 20.8011,C -0.896,E1 20.9167,E2 397.6355} C_DIS
LIN {X 78.8515,Y 108.99,Z 160,A 52.0064,B 20.8011,C -0.8977,E1 20.9125,E2 395.789} C_DIS
LIN {X 75.3194,Y 111.4601,Z 160,A 53.8561,B 20.8009,C -0.9014,E1 20.9082,E2 393.9366} C_DIS
LIN {X 71.817,Y 113.7483,Z 160,A 55.6422,B 20.8007,C -0.9044,E1 20.904,E2 392.1492} C_DIS
LIN {X 68.1215,Y 115.9992,Z 160,A 57.4597,B 20.8007,C -0.906,E1 20.8997,E2 390.3342} C_DIS
LIN {X 64.4022,Y 118.1047,Z 160,A 59.1003,B 20.8009,C -0.9004,E1 20.8957,E2 388.7151} C_DIS
LIN {X 61.7859,Y 119.495,Z 160,A 60.4679,B 20.8006,C -0.9069,E1 20.8923,E2 387.3341} C_DIS
LIN {X 58.752,Y 121.0155,Z 160,A 62.0383,B 20.8003,C -0.9143,E1 20.8884,E2 385.7479} C_DIS
LIN {X 55.3937,Y 122.5872,Z 160,A 63.4407,B 20.8006,C -0.9083,E1 20.8848,E2 384.3669} C_DIS
LIN {X 52.1268,Y 124.011,Z 160,A 64.7927,B 20.8008,C -0.9025,E1 20.8814,E2 383.035} C_DIS
LIN {X 49.5173,Y 125.0783,Z 160,A 66.1889,B 20.8004,C -0.9125,E1 20.8778,E2 381.6147} C_DIS
LIN {X 46.0117,Y 126.4079,Z 160,A 67.7757,B 20.8004,C -0.9136,E1 20.8736,E2 380.0289} C_DIS
LIN {X 43.2827,Y 127.3701,Z 160,A 69.0083,B 20.8004,C -0.9147,E1 20.8703,E2 378.7963} C_DIS
LIN {X 40.1515,Y 128.3916,Z 160,A 70.4064,B 20.8003,C -0.9156,E1 20.8666,E2 377.3988} C_DIS
LIN {X 36.6724,Y 129.4265,Z 160,A 71.9708,B 20.8002,C -0.9176,E1 20.8624,E2 375.8321} C_DIS
LIN {X 33.3751,Y 130.3153,Z 160,A 73.3035,B 20.8004,C -0.9131,E1 20.8589,E2 374.5144} C_DIS
LIN {X 30.7393,Y 130.9643,Z 160,A 74.5502,B 20.8002,C -0.9178,E1 20.8555,E2 373.2569} C_DIS
LIN {X 27.6055,Y 131.6605,Z 160,A 76.0021,B 20.8,C -0.9222,E1 20.8515,E2 371.7948} C_DIS
LIN {X 24.1383,Y 132.3384,Z 160,A 77.2837,B 20.8004,C -0.9131,E1 20.848,E2 370.5407} C_DIS
LIN {X 21.3603,Y 132.8167,Z 160,A 78.6117,B 20.8001,C -0.9191,E1 20.8443,E2 369.1975} C_DIS
LIN {X 17.6913,Y 133.3529,Z 160,A 80.2138,B 20.8001,C -0.9206,E1 20.8399,E2 367.5929} C_DIS
LIN {X 14.3994,Y 133.7483,Z 160,A 81.6085,B 20.8001,C -0.9201,E1 20.836,E2 366.2008} C_DIS
LIN {X 11.3541,Y 134.0412,Z 160,A 82.9081,B 20.8001,C -0.9201,E1 20.8324,E2 364.902} C_DIS
LIN {X 8.3032,Y 134.2647,Z 160,A 84.1962,B 20.8001,C -0.9196,E1 20.8288,E2 363.6163} C_DIS
LIN {X 5.2741,Y 134.4178,Z 160,A 85.5186,B 20.8001,C -0.9209,E1 20.8251,E2 362.2907} C_DIS
LIN {X 1.4828,Y 134.5152,Z 160,A 87.2528,B 20.7998,C -0.9259,E1 20.8202,E2 360.5427} C_DIS
LIN {X -2.2067,Y 134.5032,Z 160,A 88.6734,B 20.8001,C -0.9191,E1 20.8163,E2 359.1413} C_DIS
LIN {X -5.2741,Y 134.4178,Z 160,A 89.9838,B 20.8001,C -0.9189,E1 20.8127,E2 357.8312} C_DIS
LIN {X -8.3032,Y 134.2647,Z 160,A 91.3112,B 20.8001,C -0.92,E1 20.809,E2 356.5002} C_DIS
LIN {X -12.0875,Y 133.9792,Z 160,A 92.9384,B 20.8001,C -0.9197,E1 20.8044,E2 354.8729} C_DIS
LIN {X -15.7073,Y 133.6012,Z 160,A 94.4292,B 20.8002,C -0.9164,E1 20.8003,E2 353.3902} C_DIS
LIN {X -18.884,Y 133.1891,Z 160,A 95.8483,B 20.8002,C -0.918,E1 20.7964,E2 351.9654} C_DIS
LIN {X -22.1715,Y 132.6814,Z 160,A 97.233,B 20.8002,C -0.9157,E1 20.7926,E2 350.5856} C_DIS
LIN {X -25.2272,Y 132.1344,Z 160,A 98.5724,B 20.8002,C -0.9155,E1 20.7889,E2 349.2451} C_DIS
LIN {X -28.4212,Y 131.4844,Z 160,A 99.9659,B 20.8003,C -0.9146,E1 20.7851,E2 347.8521} C_DIS
LIN {X -31.6188,Y 130.7523,Z 160,A 101.3683,B 20.8003,C -0.9136,E1 20.7813,E2 346.4503} C_DIS
LIN {X -34.7188,Y 129.9634,Z 160,A 102.7312,B 20.8004,C -0.9123,E1 20.7776,E2 345.0885} C_DIS
LIN {X -37.8321,Y 129.0915,Z 160,A 104.1182,B 20.8004,C -0.9113,E1 20.7739,E2 343.7015} C_DIS
LIN {X -41.718,Y 127.8912,Z 160,A 105.8574,B 20.8005,C -0.9097,E1 20.7692,E2 341.9632} C_DIS
LIN {X -44.8454,Y 126.8283,Z 160,A 107.3644,B 20.8005,C -0.9122,E1 20.7652,E2 340.4454} C_DIS
LIN {X -48.3934,Y 125.5152,Z 160,A 108.7126,B 20.801,C -0.8991,E1 20.7618,E2 339.1308} C_DIS
LIN {X -51.0679,Y 124.4533,Z 160,A 110.12,B 20.8007,C -0.9051,E1 20.7581,E2 337.7027} C_DIS
LIN {X -54.1565,Y 123.1406,Z 160,A 111.6955,B 20.8005,C -0.9092,E1 20.754,E2 336.1109} C_DIS
LIN {X -57.7286,Y 121.5044,Z 160,A 113.0246,B 20.8012,C -0.8924,E1 20.7508,E2 334.8255} C_DIS
LIN {X -60.2722,Y 120.2656,Z 160,A 114.4481,B 20.8009,C -0.8996,E1 20.7472,E2 333.3769} C_DIS
LIN {X -63.6836,Y 118.4937,Z 160,A 116.1552,B 20.8009,C -0.8999,E1 20.7429,E2 331.6632} C_DIS
LIN {X -67.3818,Y 116.4305,Z 160,A 117.9753,B 20.801,C -0.8975,E1 20.7385,E2 329.8433} C_DIS
LIN {X -71.0887,Y 114.2049,Z 160,A 119.8196,B 20.8012,C -0.8943,E1 20.7341,E2 328.001} C_DIS
LIN {X -74.6759,Y 111.8922,Z 160,A 121.6545,B 20.8012,C -0.8916,E1 20.7298,E2 326.1664} C_DIS
LIN {X -78.2281,Y 109.4382,Z 160,A 123.5037,B 20.8014,C -0.8884,E1 20.7256,E2 324.3184} C_DIS
LIN {X -81.7088,Y 106.8645,Z 160,A 125.3578,B 20.8015,C -0.8851,E1 20.7215,E2 322.4655} C_DIS
LIN {X -85.1121,Y 104.1743,Z 160,A 127.2162,B 20.8017,C -0.8817,E1 20.7174,E2 320.6084} C_DIS
LIN {X -88.4594,Y 101.3474,Z 160,A 129.086,B 20.8018,C -0.8777,E1 20.7135,E2 318.7408} C_DIS
LIN {X -91.6635,Y 98.4589,Z 160,A 130.9413,B 20.802,C -0.8743,E1 20.7097,E2 316.886} C_DIS
LIN {X -94.8008,Y 95.442,Z 160,A 132.8062,B 20.8021,C -0.8705,E1 20.7059,E2 315.0224} C_DIS
LIN {X -97.8637,Y 92.2987,Z 160,A 134.6795,B 20.8023,C -0.8661,E1 20.7023,E2 313.1514} C_DIS
LIN {X -100.8985,Y 88.9713,Z 160,A 136.5817,B 20.8025,C -0.8608,E1 20.6988,E2 311.2541} C_DIS
LIN {X -103.6226,Y 85.783,Z 160,A 138.4064,B 20.8026,C -0.8578,E1 20.6955,E2 309.4274} C_DIS
LIN {X -106.3357,Y 82.3959,Z 160,A 140.2662,B 20.8028,C -0.8535,E1 20.6923,E2 307.5691} C_DIS
LIN {X -108.9329,Y 78.9301,Z 160,A 142.1222,B 20.803,C -0.8491,E1 20.6892,E2 305.7147} C_DIS
LIN {X -111.4111,Y 75.3918,Z 160,A 143.9738,B 20.8032,C -0.8446,E1 20.6863,E2 303.8646} C_DIS
LIN {X -113.7483,Y 71.817,Z 160,A 145.8113,B 20.8033,C -0.8403,E1 20.6835,E2 302.0278} C_DIS
LIN {X -115.9992,Y 68.1215,Z 160,A 147.6587,B 20.8035,C -0.8353,E1 20.6809,E2 300.1827} C_DIS
LIN {X -118.1047,Y 64.4022,Z 160,A 149.3169,B 20.804,C -0.8235,E1 20.6786,E2 298.5473} C_DIS
LIN {X -119.495,Y 61.7859,Z 160,A 150.6991,B 20.804,C -0.8248,E1 20.6768,E2 297.1526} C_DIS
LIN {X -121.0155,Y 58.752,Z 160,A 152.1538,B 20.804,C -0.8209,E1 20.675,E2 295.6991} C_DIS
LIN {X -122.6656,Y 55.2186,Z 160,A 153.8406,B 20.8042,C -0.8171,E1 20.6731,E2 294.0118} C_DIS
LIN {X -123.8074,Y 52.6144,Z 160,A 155.0444,B 20.8044,C -0.8131,E1 20.6718,E2 292.811} C_DIS
LIN {X -125.0783,Y 49.5173,Z 160,A 156.4796,B 20.8044,C -0.8092,E1 20.6703,E2 291.3771} C_DIS
LIN {X -126.2658,Y 46.4057,Z 160,A 157.996,B 20.8045,C -0.8089,E1 20.6688,E2 289.8511} C_DIS
LIN {X -127.4544,Y 43.0297,Z 160,A 159.3397,B 20.8049,C -0.797,E1 20.6676,E2 288.5319} C_DIS
LIN {X -128.4436,Y 39.9815,Z 160,A 160.7475,B 20.805,C -0.7945,E1 20.6664,E2 287.1213} C_DIS
LIN {X -129.3306,Y 37.0152,Z 160,A 162.1425,B 20.805,C -0.7935,E1 20.6653,E2 285.7191} C_DIS
LIN {X -130.188,Y 33.8768,Z 160,A 163.537,B 20.8052,C -0.7895,E1 20.6643,E2 284.3259} C_DIS
LIN {X -130.9643,Y 30.7393,Z 160,A 164.9225,B 20.8054,C -0.7856,E1 20.6634,E2 282.9416} C_DIS
LIN {X -131.6605,Y 27.6055,Z 160,A 166.4413,B 20.8053,C -0.7874,E1 20.6625,E2 281.4066} C_DIS
LIN {X -132.2776,Y 24.4783,Z 160,A 167.6648,B 20.8056,C -0.7777,E1 20.6618,E2 280.2017} C_DIS
LIN {X -132.8167,Y 21.3603,Z 160,A 169.1735,B 20.8056,C -0.78,E1 20.6611,E2 278.6756} C_DIS
LIN {X -133.3684,Y 17.5733,Z 160,A 170.6856,B 20.8059,C -0.7701,E1 20.6606,E2 277.1806} C_DIS
LIN {X -133.7456,Y 14.4246,Z 160,A 172.0197,B 20.8061,C -0.7651,E1 20.6601,E2 275.8506} C_DIS
LIN {X -134.0412,Y 11.3541,Z 160,A 173.354,B 20.8062,C -0.7618,E1 20.6598,E2 274.516} C_DIS
LIN {X -134.2725,Y 8.1779,Z 160,A 174.7344,B 20.8063,C -0.7584,E1 20.6596,E2 273.1348} C_DIS
LIN {X -134.4513,Y 4.3874,Z 160,A 176.448,B 20.8063,C -0.7572,E1 20.6594,E2 271.4121} C_DIS
LIN {X -134.5151,Y 1.4897,Z 160,A 177.6775,B 20.8065,C -0.7531,E1 20.6594,E2 270.1852} C_DIS
LIN {X -134.5032,Y -2.2067,Z 160,A 179.1647,B 20.8068,C -0.7446,E1 20.6594,E2 268.7111} C_DIS
LIN {X -134.4096,Y -5.4861,Z 160,A -179.3746,B 20.8068,C -0.7427,E1 20.6595,E2 267.2449} C_DIS
LIN {X -134.1763,Y -9.6285,Z 160,A -177.5985,B 20.807,C -0.7375,E1 20.6598,E2 265.4705} C_DIS
LIN {X -133.9025,Y -12.887,Z 160,A -176.1998,B 20.8072,C -0.7334,E1 20.6602,E2 264.0732} C_DIS
LIN {X -133.482,Y -16.7064,Z 160,A -174.581,B 20.8074,C -0.7275,E1 20.6607,E2 262.4591} C_DIS
LIN {X -132.9681,Y -20.3828,Z 160,A -172.9569,B 20.8074,C -0.7243,E1 20.6614,E2 260.8321} C_DIS
LIN {X -132.423,Y -23.6657,Z 160,A -171.5529,B 20.8076,C -0.7194,E1 20.662,E2 259.4319} C_DIS
LIN {X -131.8263,Y -26.7907,Z 160,A -170.1726,B 20.8078,C -0.7163,E1 20.6628,E2 258.0505} C_DIS
LIN {X -131.1359,Y -29.9881,Z 160,A -168.7792,B 20.8078,C -0.712,E1 20.6636,E2 256.6591} C_DIS
LIN {X -130.3953,Y -33.0597,Z 160,A -167.4209,B 20.808,C -0.7084,E1 20.6645,E2 255.3012} C_DIS
LIN {X -129.3306,Y -37.0152,Z 160,A -165.661,B 20.8082,C -0.7038,E1 20.6658,E2 253.5419} C_DIS
LIN {X -128.3916,Y -40.1515,Z 160,A -164.254,B 20.8082,C -0.7001,E1 20.667,E2 252.1353} C_DIS
LIN {X -127.201,Y -43.7707,Z 160,A -162.6108,B 20.8084,C -0.6962,E1 20.6684,E2 250.4917} C_DIS
LIN {X -126.1319,Y -46.7632,Z 160,A -161.3979,B 20.8087,C -0.6865,E1 20.6696,E2 249.2979} C_DIS
LIN {X -124.8953,Y -49.9712,Z 160,A -159.8072,B 20.8087,C -0.6874,E1 20.6712,E2 247.6936} C_DIS
LIN {X -123.7101,Y -52.8393,Z 160,A -158.5362,B 20.8089,C -0.6816,E1 20.6726,E2 246.4305} C_DIS
LIN {X -122.4531,Y -55.6937,Z 160,A -157.1031,B 20.8089,C -0.6821,E1 20.6742,E2 244.9863} C_DIS
LIN {X -121.0155,Y -58.752,Z 160,A -155.6524,B 20.8089,C -0.6785,E1 20.676,E2 243.5359} C_DIS
LIN {X -119.495,Y -61.7859,Z 160,A -154.0947,B 20.8089,C -0.6792,E1 20.678,E2 241.9662} C_DIS
LIN {X -117.4784,Y -65.539,Z 160,A -152.2723,B 20.8091,C -0.6746,E1 20.6804,E2 240.1449} C_DIS
LIN {X -115.3301,Y -69.2495,Z 160,A -150.4277,B 20.8092,C -0.6706,E1 20.683,E2 238.3002} C_DIS
LIN {X -113.0644,Y -72.8903,Z 160,A -148.5922,B 20.8093,C -0.6662,E1 20.6858,E2 236.4655} C_DIS
LIN {X -110.6708,Y -76.4756,Z 160,A -146.7431,B 20.8095,C -0.6621,E1 20.6887,E2 234.6168} C_DIS
LIN {X -108.1326,Y -80.0241,Z 160,A -144.8824,B 20.8096,C -0.6577,E1 20.6917,E2 232.7575} C_DIS
LIN {X -105.5232,Y -83.435,Z 160,A -143.0236,B 20.8096,C -0.6545,E1 20.6949,E2 230.8969} C_DIS
LIN {X -102.7755,Y -86.7971,Z 160,A -141.1638,B 20.8098,C -0.6507,E1 20.6982,E2 229.0375} C_DIS
LIN {X -99.9168,Y -90.0732,Z 160,A -139.3075,B 20.8099,C -0.6467,E1 20.7017,E2 227.1822} C_DIS
LIN {X -96.9512,Y -93.2577,Z 160,A -137.4438,B 20.81,C -0.6431,E1 20.7053,E2 225.3188} C_DIS
LIN {X -93.8832,Y -96.3457,Z 160,A -135.5733,B 20.8101,C -0.6399,E1 20.709,E2 223.4477} C_DIS
LIN {X -90.7176,Y -99.3321,Z 160,A -133.7171,B 20.8102,C -0.6363,E1 20.7128,E2 221.5924} C_DIS
LIN {X -87.4594,Y -102.2125,Z 160,A -131.8496,B 20.8103,C -0.6333,E1 20.7167,E2 219.7243} C_DIS
LIN {X -84.1141,Y -104.9827,Z 160,A -129.9915,B 20.8104,C -0.6302,E1 20.7207,E2 217.8663} C_DIS
LIN {X -80.6625,Y -107.6572,Z 160,A -128.1324,B 20.8105,C -0.6269,E1 20.7249,E2 216.0084} C_DIS
LIN {X -77.1847,Y -110.1774,Z 160,A -126.2823,B 20.8105,C -0.6247,E1 20.7291,E2 214.1567} C_DIS
LIN {X -73.6125,Y -112.5955,Z 160,A -124.4518,B 20.8107,C -0.6215,E1 20.7333,E2 212.3279} C_DIS
LIN {X -69.9768,Y -114.8903,Z 160,A -122.6086,B 20.8107,C -0.6192,E1 20.7377,E2 210.484} C_DIS
LIN {X -66.2609,Y -117.0727,Z 160,A -120.7752,B 20.8108,C -0.6166,E1 20.7422,E2 208.6515} C_DIS
LIN {X -63.2927,Y -118.7038,Z 160,A -119.4227,B 20.811,C -0.6108,E1 20.7455,E2 207.3107} C_DIS
LIN {X -59.8115,Y -120.4928,Z 160,A -117.793,B 20.811,C -0.6071,E1 20.7495,E2 205.6861} C_DIS
LIN {X -57.0453,Y -121.8281,Z 160,A -116.3452,B 20.811,C -0.6115,E1 20.7532,E2 204.2212} C_DIS
LIN {X -54.1565,Y -123.1406,Z 160,A -115.0869,B 20.8111,C -0.606,E1 20.7564,E2 202.9748} C_DIS
LIN {X -51.0679,Y -124.4533,Z 160,A -113.522,B 20.811,C -0.6104,E1 20.7605,E2 201.3933} C_DIS
LIN {X -47.4217,Y -125.8853,Z 160,A -112.2043,B 20.8114,C -0.5936,E1 20.7638,E2 200.1193} C_DIS
LIN {X -44.8454,Y -126.8283,Z 160,A -110.8151,B 20.8112,C -0.6021,E1 20.7675,E2 198.7029} C_DIS
LIN {X -41.718,Y -127.8912,Z 160,A -109.2594,B 20.8111,C -0.6074,E1 20.7717,E2 197.1286} C_DIS
LIN {X -37.9601,Y -129.054,Z 160,A -107.7763,B 20.8113,C -0.5979,E1 20.7756,E2 195.6693} C_DIS
LIN {X -34.871,Y -129.9228,Z 160,A -106.5893,B 20.8116,C -0.5891,E1 20.7787,E2 194.5047} C_DIS
LIN {X -32.3078,Y -130.5862,Z 160,A -105.2359,B 20.8113,C -0.5983,E1 20.7824,E2 193.1231} C_DIS
LIN {X -28.7449,Y -131.4145,Z 160,A -103.6765,B 20.8113,C -0.5976,E1 20.7867,E2 191.5633} C_DIS
LIN {X -26.0409,Y -131.9788,Z 160,A -102.5025,B 20.8113,C -0.5969,E1 20.7899,E2 190.3895} C_DIS
LIN {X -22.918,Y -132.5568,Z 160,A -101.1506,B 20.8113,C -0.5964,E1 20.7936,E2 189.0375} C_DIS
LIN {X -19.3226,Y -133.1265,Z 160,A -99.5612,B 20.8113,C -0.5977,E1 20.798,E2 187.4427} C_DIS
LIN {X -15.9024,Y -133.5779,Z 160,A -98.1472,B 20.8114,C -0.595,E1 20.8019,E2 186.0352} C_DIS
LIN {X -12.887,Y -133.9025,Z 160,A -96.8453,B 20.8114,C -0.5952,E1 20.8055,E2 184.7316} C_DIS
LIN {X -9.7627,Y -134.1665,Z 160,A -95.524,B 20.8114,C -0.5946,E1 20.8092,E2 183.4115} C_DIS
LIN {X -6.6229,Y -134.3582,Z 160,A -94.1055,B 20.8114,C -0.5981,E1 20.8132,E2 181.9826} C_DIS
LIN {X -2.4439,Y -134.4993,Z 160,A -92.36,B 20.8114,C -0.5967,E1 20.8181,E2 180.2408} C_DIS
LIN {X 0.9519,Y -134.5171,Z 160,A -91.0295,B 20.8114,C -0.5918,E1 20.8217,E2 178.924} C_DIS
Enddeposition()
LIN {X 0.9519,Y -134.5171,Z 160,A -91.0295,B 20.8114,C -0.5918,E1 20.8217,E2 178.924} C_DIS
Startdeposition()
$VEL.CP = VEL_PRINT
LIN {X -0.4093,Y -133.5952,Z 160,A -91.8526,B 19.655,C -0.4202,E1 19.6581,E2 180.1363} C_DIS
LIN {X -4.4308,Y -133.5238,Z 160,A -93.6573,B 19.655,C -0.4167,E1 19.653,E2 181.9516} C_DIS
LIN {X -8.4596,Y -133.3274,Z 160,A -95.2607,B 19.655,C -0.4219,E1 19.6486,E2 183.5402} C_DIS
LIN {X -12.7255,Y -132.9878,Z 160,A -97.1096,B 19.655,C -0.4215,E1 19.6434,E2 185.3914} C_DIS
LIN {X -16.7974,Y -132.5362,Z 160,A -98.9075,B 19.655,C -0.4201,E1 19.6384,E2 187.1949} C_DIS
LIN {X -20.3488,Y -132.0364,Z 160,A -100.3616,B 19.655,C -0.424,E1 19.6345,E2 188.6392} C_DIS
LIN {X -23.7575,Y -131.4659,Z 160,A -101.8827,B 19.655,C -0.4229,E1 19.6303,E2 190.1654} C_DIS
LIN {X -27.8298,Y -130.6648,Z 160,A -103.6698,B 19.655,C -0.4234,E1 19.6254,E2 191.9536} C_DIS
LIN {X -31.4475,Y -129.8411,Z 160,A -105.1355,B 19.6548,C -0.4293,E1 19.6214,E2 193.4041} C_DIS
LIN {X -35.5306,Y -128.7844,Z 160,A -107.1005,B 19.6549,C -0.4241,E1 19.6161,E2 195.3884} C_DIS
LIN {X -39.0747,Y -127.7529,Z 160,A -108.6509,B 19.6549,C -0.4266,E1 19.6119,E2 196.9349} C_DIS
LIN {X -42.9465,Y -126.5062,Z 160,A -110.5388,B 19.6549,C -0.4222,E1 19.6069,E2 198.8403} C_DIS
LIN {X -46.7206,Y -125.1591,Z 160,A -112.0725,B 19.6548,C -0.4312,E1 19.6029,E2 200.3513} C_DIS
LIN {X -49.7929,Y -123.9689,Z 160,A -113.4087,B 19.6547,C -0.4356,E1 19.5995,E2 201.6781} C_DIS
LIN {X -52.3336,Y -122.92,Z 160,A -114.8152,B 19.6548,C -0.4278,E1 19.5958,E2 203.1122} C_DIS
LIN {X -55.7844,Y -121.391,Z 160,A -116.3386,B 19.6548,C -0.4334,E1 19.5919,E2 204.6237} C_DIS
LIN {X -58.8699,Y -119.9249,Z 160,A -117.7969,B 19.6547,C -0.4354,E1 19.5882,E2 206.0808} C_DIS
LIN {X -61.9922,Y -118.3408,Z 160,A -119.2502,B 19.6546,C -0.4392,E1 19.5847,E2 207.5278} C_DIS
LIN {X -65.4173,Y -116.4847,Z 160,A -121.0538,B 19.6546,C -0.4362,E1 19.5802,E2 209.3472} C_DIS
LIN {X -69.0969,Y -114.3404,Z 160,A -122.8835,B 19.6546,C -0.4387,E1 19.5758,E2 211.1766} C_DIS
LIN {X -72.6934,Y -112.0882,Z 160,A -124.7455,B 19.6546,C -0.4399,E1 19.5714,E2 213.043} C_DIS
LIN {X -76.3173,Y -109.653,Z 160,A -126.5926,B 19.6545,C -0.4439,E1 19.5672,E2 214.8862} C_DIS
LIN {X -79.8429,Y -107.1131,Z 160,A -128.4819,B 19.6545,C -0.4461,E1 19.5629,E2 216.7777} C_DIS
LIN {X -83.3099,Y -104.4394,Z 160,A -130.2784,B 19.6543,C -0.4526,E1 19.559,E2 218.5632} C_DIS
LIN {X -86.5508,Y -101.7696,Z 160,A -132.184,B 19.6543,C -0.4519,E1 19.5549,E2 220.4804} C_DIS
LIN {X -89.8766,Y -98.8449,Z 160,A -134.085,B 19.6543,C -0.4556,E1 19.5509,E2 222.3804} C_DIS
LIN {X -93.1849,Y -95.733,Z 160,A -136.0749,B 19.6542,C -0.4579,E1 19.5469,E2 224.3741} C_DIS
LIN {X -96.3049,Y -92.5939,Z 160,A -137.9908,B 19.6542,C -0.4612,E1 19.5431,E2 226.2907} C_DIS
LIN {X -99.2853,Y -89.3905,Z 160,A -139.6308,B 19.6538,C -0.4744,E1 19.5401,E2 227.9007} C_DIS
LIN {X -101.6518,Y -86.6894,Z 160,A -141.4252,B 19.6539,C -0.4682,E1 19.5368,E2 229.7244} C_DIS
LIN {X -104.436,Y -83.3142,Z 160,A -143.1006,B 19.6537,C -0.4802,E1 19.5339,E2 231.374} C_DIS
LIN {X -106.5758,Y -80.5587,Z 160,A -144.7831,B 19.6537,C -0.4767,E1 19.531,E2 233.0775} C_DIS
LIN {X -109.0349,Y -77.1982,Z 160,A -146.6193,B 19.6537,C -0.4791,E1 19.528,E2 234.9182} C_DIS
LIN {X -111.9226,Y -72.9485,Z 160,A -148.8115,B 19.6536,C -0.4851,E1 19.5246,E2 237.1068} C_DIS
LIN {X -114.232,Y -69.2761,Z 160,A -150.6712,B 19.6534,C -0.4899,E1 19.5218,E2 238.9644} C_DIS
LIN {X -116.244,Y -65.8453,Z 160,A -152.4434,B 19.6534,C -0.4919,E1 19.5194,E2 240.7428} C_DIS
LIN {X -118.2589,Y -62.1482,Z 160,A -154.0049,B 19.653,C -0.506,E1 19.5173,E2 242.2729} C_DIS
LIN {X -119.9768,Y -58.7646,Z 160,A -155.9559,B 19.6532,C -0.4982,E1 19.5149,E2 244.2608} C_DIS
LIN {X -121.8609,Y -54.7499,Z 160,A -157.692,B 19.653,C -0.5098,E1 19.5129,E2 245.9748} C_DIS
LIN {X -123.1499,Y -51.7862,Z 160,A -159.1214,B 19.6529,C -0.512,E1 19.5113,E2 247.4078} C_DIS
LIN {X -124.5228,Y -48.3907,Z 160,A -160.7858,B 19.6529,C -0.513,E1 19.5096,E2 249.0815} C_DIS
LIN {X -126.1349,Y -44.0191,Z 160,A -162.6661,B 19.6526,C -0.5232,E1 19.5078,E2 250.9451} C_DIS
LIN {X -127.2701,Y -40.6195,Z 160,A -164.1857,B 19.6525,C -0.5284,E1 19.5065,E2 252.4605} C_DIS
LIN {X -128.2813,Y -37.3042,Z 160,A -165.7772,B 19.6525,C -0.5288,E1 19.5052,E2 254.0626} C_DIS
LIN {X -129.4497,Y -33.0219,Z 160,A -167.6894,B 19.6523,C -0.5342,E1 19.5038,E2 255.9733} C_DIS
LIN {X -130.9424,Y -26.4909,Z 160,A -170.5551,B 19.6521,C -0.5432,E1 19.5021,E2 258.8342} C_DIS
LIN {X -131.6724,Y -22.5926,Z 160,A -172.3557,B 19.6521,C -0.5446,E1 19.5012,E2 260.6444} C_DIS
LIN {X -132.3794,Y -17.9938,Z 160,A -174.6575,B 19.6521,C -0.5394,E1 19.5003,E2 262.9797} C_DIS
LIN {X -132.8146,Y -14.4219,Z 160,A -175.8446,B 19.6517,C -0.5574,E1 19.4999,E2 264.1222} C_DIS
LIN {X -133.1993,Y -10.2949,Z 160,A -177.7059,B 19.6517,C -0.5598,E1 19.4995,E2 265.9908} C_DIS
LIN {X -133.4305,Y -6.6343,Z 160,A -179.1952,B 19.6514,C -0.5679,E1 19.4992,E2 267.4678} C_DIS
LIN {X -133.5679,Y -2.7658,Z 160,A 179.1617,B 19.6513,C -0.5737,E1 19.4992,E2 269.1065} C_DIS
LIN {X -133.5923,Y 1.0161,Z 160,A 177.3409,B 19.6513,C -0.5714,E1 19.4992,E2 270.9484} C_DIS
LIN {X -133.4965,Y 5.1389,Z 160,A 175.6802,B 19.6511,C -0.581,E1 19.4992,E2 272.5935} C_DIS
LIN {X -133.3091,Y 8.7581,Z 160,A 174.1452,B 19.6509,C -0.5866,E1 19.4995,E2 274.1239} C_DIS
LIN {X -132.9768,Y 12.8404,Z 160,A 172.4624,B 19.6507,C -0.5948,E1 19.4999,E2 275.7951} C_DIS
LIN {X -132.7203,Y 15.275,Z 160,A 171.0617,B 19.6509,C -0.5851,E1 19.5004,E2 277.2359} C_DIS
LIN {X -132.0882,Y 20.0145,Z 160,A 169.2618,B 19.6505,C -0.6008,E1 19.5011,E2 279.0028} C_DIS
LIN {X -131.0753,Y 25.8362,Z 160,A 165.8743,B 19.6512,C -0.5773,E1 19.5029,E2 282.487} C_DIS
LIN {X -129.8351,Y 31.4723,Z 160,A 164.1643,B 19.6501,C -0.6131,E1 19.5039,E2 284.1029} C_DIS
LIN {X -128.8623,Y 35.252,Z 160,A 162.3912,B 19.6501,C -0.6145,E1 19.5052,E2 285.8852} C_DIS
LIN {X -127.7989,Y 38.9243,Z 160,A 160.7809,B 19.6499,C -0.6206,E1 19.5064,E2 287.4893} C_DIS
LIN {X -126.4628,Y 43.0731,Z 160,A 158.9247,B 19.6497,C -0.6268,E1 19.5081,E2 289.341} C_DIS
LIN {X -125.1903,Y 46.6375,Z 160,A 157.2856,B 19.6496,C -0.6311,E1 19.5096,E2 290.9793} C_DIS
LIN {X -123.9715,Y 49.7863,Z 160,A 156.0142,B 19.6492,C -0.642,E1 19.5109,E2 292.2274} C_DIS
LIN {X -121.8867,Y 54.6922,Z 160,A 153.9487,B 19.6488,C -0.6569,E1 19.5132,E2 294.2631} C_DIS
LIN {X -117.8979,Y 62.8357,Z 160,A 149.5429,B 19.649,C -0.6486,E1 19.5187,E2 298.7246} C_DIS
LIN {X -115.8349,Y 66.5624,Z 160,A 147.6667,B 19.649,C -0.6519,E1 19.5212,E2 300.6038} C_DIS
LIN {X -114.1138,Y 69.4714,Z 160,A 146.1572,B 19.6489,C -0.6537,E1 19.5234,E2 302.1181} C_DIS
LIN {X -111.5389,Y 73.5335,Z 160,A 144.3285,B 19.6484,C -0.6681,E1 19.5261,E2 303.916} C_DIS
LIN {X -109.1659,Y 77.0123,Z 160,A 142.3913,B 19.6484,C -0.668,E1 19.5292,E2 305.866} C_DIS
LIN {X -106.6129,Y 80.5096,Z 160,A 140.5238,B 19.6483,C -0.6724,E1 19.5323,E2 307.7319} C_DIS
LIN {X -104.1193,Y 83.7098,Z 160,A 138.7025,B 19.6483,C -0.6738,E1 19.5355,E2 309.5602} C_DIS
LIN {X -101.1524,Y 87.2715,Z 160,A 136.7358,B 19.648,C -0.6796,E1 19.539,E2 311.5215} C_DIS
LIN {X -95.5957,Y 93.3255,Z 160,A 132.417,B 19.6487,C -0.6583,E1 19.5475,E2 315.9285} C_DIS
LIN {X -91.2191,Y 97.6076,Z 160,A 130.6421,B 19.6475,C -0.6961,E1 19.5509,E2 317.5997} C_DIS
LIN {X -88.7633,Y 99.8458,Z 160,A 128.9032,B 19.6478,C -0.6874,E1 19.5546,E2 319.3737} C_DIS
LIN {X -86.3148,Y 101.9702,Z 160,A 127.8374,B 19.6472,C -0.7027,E1 19.5567,E2 320.3994} C_DIS
LIN {X -81.7722,Y 105.6476,Z 160,A 125.188,B 19.6472,C -0.7024,E1 19.5626,E2 323.0624} C_DIS
LIN {X -79.1789,Y 107.6049,Z 160,A 123.7455,B 19.6472,C -0.7033,E1 19.5658,E2 324.5089} C_DIS
LIN {X -75.2877,Y 110.363,Z 160,A 121.6881,B 19.6471,C -0.7068,E1 19.5705,E2 326.5651} C_DIS
LIN {X -71.6162,Y 112.7801,Z 160,A 119.7942,B 19.647,C -0.7099,E1 19.5749,E2 328.4577} C_DIS
LIN {X -67.7823,Y 115.1247,Z 160,A 117.9234,B 19.6468,C -0.7154,E1 19.5794,E2 330.3195} C_DIS
LIN {X -63.7074,Y 117.429,Z 160,A 115.6438,B 19.647,C -0.7083,E1 19.585,E2 332.6289} C_DIS
LIN {X -60.843,Y 118.936,Z 160,A 114.5961,B 19.6465,C -0.7236,E1 19.5875,E2 333.6347} C_DIS
LIN {X -57.9211,Y 120.3863,Z 160,A 113.1425,B 19.6465,C -0.7236,E1 19.5912,E2 335.0932} C_DIS
LIN {X -55.0395,Y 121.7314,Z 160,A 111.7624,B 19.6465,C -0.7249,E1 19.5947,E2 336.4739} C_DIS
LIN {X -51.9709,Y 123.0727,Z 160,A 110.0644,B 19.6467,C -0.7167,E1 19.5991,E2 338.2014} C_DIS
LIN {X -48.94,Y 124.3093,Z 160,A 108.9258,B 19.6463,C -0.7288,E1 19.602,E2 339.3071} C_DIS
LIN {X -45.7714,Y 125.5102,Z 160,A 107.4611,B 19.6463,C -0.7301,E1 19.6058,E2 340.7717} C_DIS
LIN {X -41.6011,Y 126.9542,Z 160,A 105.1465,B 19.6468,C -0.7159,E1 19.6121,E2 343.1344} C_DIS
LIN {X -37.8079,Y 128.1338,Z 160,A 103.9008,B 19.6461,C -0.7355,E1 19.6153,E2 344.3244} C_DIS
LIN {X -34.3321,Y 129.1083,Z 160,A 102.3316,B 19.6461,C -0.7362,E1 19.6195,E2 345.8948} C_DIS
LIN {X -30.4815,Y 130.0734,Z 160,A 100.2275,B 19.6466,C -0.7219,E1 19.6254,E2 348.0451} C_DIS
LIN {X -26.8967,Y 130.8598,Z 160,A 99.0463,B 19.646,C -0.7386,E1 19.6285,E2 349.1784} C_DIS
LIN {X -24.0736,Y 131.4094,Z 160,A 97.664,B 19.6462,C -0.7336,E1 19.6323,E2 350.5775} C_DIS
LIN {X -19.607,Y 132.1505,Z 160,A 95.7978,B 19.646,C -0.7378,E1 19.6374,E2 352.4334} C_DIS
LIN {X -16.0709,Y 132.6253,Z 160,A 94.3354,B 19.6459,C -0.7413,E1 19.6414,E2 353.8867} C_DIS
LIN {X -12.744,Y 132.986,Z 160,A 92.8982,B 19.6459,C -0.7419,E1 19.6454,E2 355.3232} C_DIS
LIN {X -8.7252,Y 133.3111,Z 160,A 91.0979,B 19.6459,C -0.7397,E1 19.6505,E2 357.1309} C_DIS
LIN {X -4.9299,Y 133.5047,Z 160,A 89.4381,B 19.6459,C -0.7389,E1 19.6551,E2 358.7934} C_DIS
LIN {X -0.8519,Y 133.5927,Z 160,A 87.7429,B 19.6459,C -0.7414,E1 19.6598,E2 360.4812} C_DIS
LIN {X 3.4279,Y 133.5517,Z 160,A 85.9688,B 19.6458,C -0.7441,E1 19.6647,E2 362.2471} C_DIS
LIN {X 6.8483,Y 133.4198,Z 160,A 84.4843,B 19.6458,C -0.7434,E1 19.6689,E2 363.7329} C_DIS
LIN {X 10.8753,Y 133.1524,Z 160,A 82.7147,B 19.6458,C -0.7417,E1 19.6738,E2 365.5066} C_DIS
LIN {X 14.511,Y 132.805,Z 160,A 81.1228,B 19.6459,C -0.7404,E1 19.6783,E2 367.1009} C_DIS
LIN {X 18.6246,Y 132.2909,Z 160,A 79.3756,B 19.6459,C -0.7412,E1 19.6831,E2 368.8441} C_DIS
LIN {X 22.3518,Y 131.7126,Z 160,A 77.6807,B 19.646,C -0.7374,E1 19.6878,E2 370.5477} C_DIS
LIN {X 26.8084,Y 130.8778,Z 160,A 75.8159,B 19.646,C -0.7398,E1 19.6929,E2 372.4027} C_DIS
LIN {X 30.3196,Y 130.1104,Z 160,A 74.1539,B 19.6461,C -0.734,E1 19.6974,E2 374.0789} C_DIS
LIN {X 34.3572,Y 129.1016,Z 160,A 72.5307,B 19.6459,C -0.7395,E1 19.7018,E2 375.6825} C_DIS
LIN {X 38.0212,Y 128.0713,Z 160,A 70.9166,B 19.6459,C -0.739,E1 19.7061,E2 377.2944} C_DIS
LIN {X 41.6613,Y 126.9341,Z 160,A 69.1812,B 19.6462,C -0.7336,E1 19.7107,E2 379.0418} C_DIS
LIN {X 45.2783,Y 125.688,Z 160,A 67.6786,B 19.646,C -0.7378,E1 19.7147,E2 380.5278} C_DIS
LIN {X 47.958,Y 124.691,Z 160,A 66.4923,B 19.646,C -0.7382,E1 19.7177,E2 381.7095} C_DIS
LIN {X 51.1508,Y 123.4152,Z 160,A 64.9317,B 19.6462,C -0.7331,E1 19.7218,E2 383.2805} C_DIS
LIN {X 54.3531,Y 122.0384,Z 160,A 63.44,B 19.6462,C -0.7316,E1 19.7256,E2 384.7721} C_DIS
LIN {X 56.9813,Y 120.8353,Z 160,A 62.107,B 19.6464,C -0.7262,E1 19.729,E2 386.1166} C_DIS
LIN {X 60.1104,Y 119.309,Z 160,A 60.755,B 19.6463,C -0.7302,E1 19.7324,E2 387.452} C_DIS
LIN {X 63.6321,Y 117.47,Z 160,A 58.9274,B 19.6465,C -0.7227,E1 19.7369,E2 389.2951} C_DIS
LIN {X 69.5346,Y 114.0754,Z 160,A 55.9906,B 19.6467,C -0.7178,E1 19.744,E2 392.2348} C_DIS
LIN {X 73.3812,Y 111.6392,Z 160,A 54.099,B 19.6467,C -0.7172,E1 19.7484,E2 394.1199} C_DIS
LIN {X 76.9736,Y 109.1933,Z 160,A 52.2439,B 19.6468,C -0.7145,E1 19.7527,E2 395.9748} C_DIS
LIN {X 80.582,Y 106.5583,Z 160,A 50.5402,B 19.6466,C -0.7202,E1 19.7564,E2 397.6539} C_DIS
LIN {X 83.416,Y 104.3549,Z 160,A 48.8121,B 19.647,C -0.7093,E1 19.7603,E2 399.4055} C_DIS
LIN {X 86.5962,Y 101.7311,Z 160,A 47.3073,B 19.6467,C -0.7172,E1 19.7635,E2 400.8796} C_DIS
LIN {X 88.6785,Y 99.9214,Z 160,A 45.8456,B 19.6472,C -0.703,E1 19.7666,E2 402.3757} C_DIS
LIN {X 91.9825,Y 96.8891,Z 160,A 43.9139,B 19.6474,C -0.6987,E1 19.7705,E2 404.3098} C_DIS
LIN {X 95.0226,Y 93.9091,Z 160,A 42.1058,B 19.6474,C -0.6956,E1 19.7741,E2 406.1171} C_DIS
LIN {X 97.3686,Y 91.4742,Z 160,A 40.675,B 19.6476,C -0.6933,E1 19.7769,E2 407.5467} C_DIS
LIN {X 100.2159,Y 88.3454,Z 160,A 38.9019,B 19.6476,C -0.691,E1 19.7802,E2 409.3162} C_DIS
LIN {X 103.1276,Y 84.929,Z 160,A 36.9363,B 19.6478,C -0.6848,E1 19.7837,E2 411.2883} C_DIS
LIN {X 105.925,Y 81.4131,Z 160,A 35.0126,B 19.648,C -0.6804,E1 19.787,E2 413.2133} C_DIS
LIN {X 108.6676,Y 77.7139,Z 160,A 33.1277,B 19.648,C -0.6794,E1 19.7901,E2 415.0892} C_DIS
LIN {X 111.0035,Y 74.3395,Z 160,A 31.3238,B 19.6482,C -0.6731,E1 19.7929,E2 416.9001} C_DIS
LIN {X 113.5023,Y 70.4653,Z 160,A 29.3847,B 19.6483,C -0.6697,E1 19.7958,E2 418.8366} C_DIS
LIN {X 115.8183,Y 66.5912,Z 160,A 27.4151,B 19.6486,C -0.6631,E1 19.7986,E2 420.8125} C_DIS
LIN {X 117.9648,Y 62.7084,Z 160,A 25.5425,B 19.6486,C -0.6593,E1 19.8011,E2 422.6834} C_DIS
LIN {X 120.0189,Y 58.6794,Z 160,A 23.5664,B 19.6489,C -0.6524,E1 19.8036,E2 424.6661} C_DIS
LIN {X 121.7616,Y 54.972,Z 160,A 21.9353,B 19.6489,C -0.653,E1 19.8055,E2 426.2841} C_DIS
LIN {X 123.3048,Y 51.4153,Z 160,A 20.3609,B 19.6489,C -0.6522,E1 19.8072,E2 427.8496} C_DIS
LIN {X 124.4818,Y 48.4963,Z 160,A 18.9976,B 19.6491,C -0.6477,E1 19.8086,E2 429.2163} C_DIS
LIN {X 125.602,Y 45.517,Z 160,A 17.606,B 19.6492,C -0.6426,E1 19.81,E2 430.6128} C_DIS
LIN {X 127.5822,Y 39.6322,Z 160,A 14.958,B 19.6494,C -0.6354,E1 19.8123,E2 433.2626} C_DIS
LIN {X 128.6402,Y 36.0462,Z 160,A 13.4124,B 19.6495,C -0.6332,E1 19.8135,E2 434.8032} C_DIS
LIN {X 129.4803,Y 32.9011,Z 160,A 12.0682,B 19.6495,C -0.6313,E1 19.8144,E2 436.1429} C_DIS
LIN {X 130.3091,Y 29.4496,Z 160,A 10.2807,B 19.6501,C -0.615,E1 19.8156,E2 437.9649} C_DIS
LIN {X 131.3925,Y 24.1681,Z 160,A 8.106,B 19.6501,C -0.614,E1 19.8167,E2 440.126} C_DIS
LIN {X 132.038,Y 20.3383,Z 160,A 6.5688,B 19.6501,C -0.6145,E1 19.8174,E2 441.6499} C_DIS
LIN {X 132.5798,Y 16.4523,Z 160,A 4.8283,B 19.6503,C -0.6068,E1 19.818,E2 443.4} C_DIS
LIN {X 132.9792,Y 12.8157,Z 160,A 3.3229,B 19.6503,C -0.6047,E1 19.8185,E2 444.8998} C_DIS
LIN {X 133.2945,Y 8.9908,Z 160,A 1.5703,B 19.6507,C -0.5948,E1 19.8188,E2 446.668} C_DIS
LIN {X 133.4992,Y 5.0698,Z 160,A 0.0097,B 19.6507,C -0.595,E1 19.819,E2 448.2159} C_DIS
LIN {X 133.5938,Y 0.7949,Z 160,A -1.7442,B 19.6507,C -0.5928,E1 19.819,E2 449.9629} C_DIS
LIN {X 133.5629,Y -3.0262,Z 160,A -3.5836,B 19.6511,C -0.5787,E1 19.819,E2 451.8294} C_DIS
LIN {X 133.3678,Y -7.8039,Z 160,A -5.4598,B 19.6511,C -0.58,E1 19.8188,E2 453.6874} C_DIS
LIN {X 133.1014,Y -11.4795,Z 160,A -7.024,B 19.6512,C -0.5758,E1 19.8184,E2 455.252} C_DIS
LIN {X 132.6921,Y -15.5114,Z 160,A -8.8068,B 19.6514,C -0.5683,E1 19.8179,E2 457.043} C_DIS
LIN {X 132.1328,Y -19.7259,Z 160,A -10.6171,B 19.6516,C -0.5631,E1 19.8172,E2 458.8547} C_DIS
LIN {X 131.4134,Y -24.0514,Z 160,A -12.3917,B 19.6516,C -0.562,E1 19.8163,E2 460.6192} C_DIS
LIN {X 130.8443,Y -26.9732,Z 160,A -13.8054,B 19.6519,C -0.5519,E1 19.8155,E2 462.0517} C_DIS
LIN {X 129.9268,Y -31.092,Z 160,A -15.4791,B 19.6519,C -0.5523,E1 19.8145,E2 463.7117} C_DIS
LIN {X 129.1094,Y -34.3279,Z 160,A -16.8873,B 19.6519,C -0.5489,E1 19.8135,E2 465.1193} C_DIS
LIN {X 128.186,Y -37.6296,Z 160,A -18.2389,B 19.6519,C -0.5497,E1 19.8125,E2 466.4586} C_DIS
LIN {X 127.0873,Y -41.1918,Z 160,A -20.0443,B 19.6523,C -0.5356,E1 19.8109,E2 468.292} C_DIS
LIN {X 125.8639,Y -44.7904,Z 160,A -21.4354,B 19.6521,C -0.5413,E1 19.8097,E2 469.6564} C_DIS
LIN {X 124.5732,Y -48.2611,Z 160,A -23.1388,B 19.6524,C -0.5314,E1 19.808,E2 471.3765} C_DIS
LIN {X 123.187,Y -51.6972,Z 160,A -24.7288,B 19.6525,C -0.5266,E1 19.8063,E2 472.9691} C_DIS
LIN {X 121.4828,Y -55.5859,Z 160,A -26.4609,B 19.6525,C -0.5252,E1 19.8044,E2 474.6933} C_DIS
LIN {X 119.9663,Y -58.786,Z 160,A -28.2015,B 19.6529,C -0.511,E1 19.8022,E2 476.4636} C_DIS
LIN {X 117.7599,Y -63.0931,Z 160,A -30.397,B 19.6532,C -0.4998,E1 19.7993,E2 478.6771} C_DIS
LIN {X 116.115,Y -66.0715,Z 160,A -31.6089,B 19.653,C -0.5065,E1 19.7977,E2 479.8609} C_DIS
LIN {X 113.8427,Y -69.9138,Z 160,A -33.4831,B 19.6531,C -0.5029,E1 19.795,E2 481.7332} C_DIS
LIN {X 112.2275,Y -72.4789,Z 160,A -35.2804,B 19.6537,C -0.4776,E1 19.7922,E2 483.5935} C_DIS
LIN {X 109.6272,Y -76.3543,Z 160,A -36.7699,B 19.6533,C -0.4946,E1 19.7899,E2 485.0234} C_DIS
LIN {X 107.0316,Y -79.9524,Z 160,A -38.6747,B 19.6534,C -0.4894,E1 19.7868,E2 486.9313} C_DIS
LIN {X 104.5661,Y -83.1507,Z 160,A -40.7249,B 19.6539,C -0.4711,E1 19.7832,E2 489.0232} C_DIS
LIN {X 102.0963,Y -86.1656,Z 160,A -42.2068,B 19.6538,C -0.4751,E1 19.7805,E2 490.4844} C_DIS
LIN {X 98.6935,Y -90.0435,Z 160,A -44.2614,B 19.6538,C -0.4765,E1 19.7767,E2 492.5229} C_DIS
LIN {X 95.7262,Y -93.1919,Z 160,A -46.091,B 19.6538,C -0.4732,E1 19.7732,E2 494.3519} C_DIS
LIN {X 92.4991,Y -96.3954,Z 160,A -48.1271,B 19.654,C -0.4649,E1 19.7691,E2 496.4014} C_DIS
LIN {X 88.8591,Y -99.7612,Z 160,A -50.1768,B 19.654,C -0.4635,E1 19.7649,E2 498.4447} C_DIS
LIN {X 85.5094,Y -102.647,Z 160,A -52.0745,B 19.6541,C -0.4593,E1 19.7608,E2 500.3452} C_DIS
LIN {X 82.9414,Y -104.7327,Z 160,A -53.3278,B 19.6541,C -0.4634,E1 19.7581,E2 501.58} C_DIS
LIN {X 79.2504,Y -107.5523,Z 160,A -55.4417,B 19.6543,C -0.4541,E1 19.7534,E2 503.7116} C_DIS
LIN {X 75.5786,Y -110.1634,Z 160,A -57.3264,B 19.6543,C -0.4524,E1 19.7491,E2 505.5929} C_DIS
LIN {X 73.3508,Y -111.6592,Z 160,A -58.9369,B 19.6548,C -0.4305,E1 19.7452,E2 507.2611} C_DIS
LIN {X 69.5527,Y -114.0643,Z 160,A -60.4414,B 19.6545,C -0.4451,E1 19.7417,E2 508.7162} C_DIS
LIN {X 65.9133,Y -116.2052,Z 160,A -62.3385,B 19.6546,C -0.4383,E1 19.7371,E2 510.6261} C_DIS
LIN {X 61.422,Y -118.6402,Z 160,A -64.4782,B 19.6546,C -0.4369,E1 19.7318,E2 512.762} C_DIS
LIN {X 58.4537,Y -120.1302,Z 160,A -66.0735,B 19.6548,C -0.4274,E1 19.7278,E2 514.3798} C_DIS
LIN {X 55.2632,Y -121.6313,Z 160,A -67.3316,B 19.6547,C -0.4359,E1 19.7247,E2 515.6085} C_DIS
LIN {X 52.1505,Y -122.9977,Z 160,A -68.7827,B 19.6547,C -0.4342,E1 19.7209,E2 517.0603} C_DIS
LIN {X 49.0332,Y -124.2731,Z 160,A -70.229,B 19.6547,C -0.4322,E1 19.7172,E2 518.5083} C_DIS
LIN {X 45.4729,Y -125.6179,Z 160,A -71.7273,B 19.6547,C -0.4358,E1 19.7133,E2 519.9917} C_DIS
LIN {X 39.9309,Y -127.49,Z 160,A -74.3309,B 19.6548,C -0.4288,E1 19.7064,E2 522.6095} C_DIS
LIN {X 36.2558,Y -128.5816,Z 160,A -75.9428,B 19.6548,C -0.4285,E1 19.702,E2 524.2187} C_DIS
LIN {X 32.2083,Y -129.6562,Z 160,A -77.7722,B 19.6548,C -0.4253,E1 19.6971,E2 526.0539} C_DIS
Enddeposition()
END
